// ---- GlobalTextList.TcGTLO
TEXTLIST GlobalTextList
  6525 = ' '
  3937 = '      Suction'
  4564 = '     KR5 Magnet'
  5885 = '     Magnet'
  1846 = ' Suction'
  271 = '%s'
  243 = '+'
  1867 = '-'
  4558 = '1-100'
  645 = '10'
  4817 = '100-200'
  551 = '1000'
  201 = '1001'
  301 = '1002'
  663 = '1003'
  224 = '1004'
  174 = '1005'
  178 = '1006'
  933 = '1007'
  532 = '1008'
  34 = '1027'
  349 = '1028'
  986 = '1029'
  837 = '1030'
  751 = '1031'
  65 = '1032'
  93 = '1033'
  410 = '1034'
  763 = '1035'
  289 = '1036'
  454 = '1037'
  54 = '1038'
  692 = '1039'
  219 = '1040'
  822 = '1041'
  60 = '1042'
  614 = '1222'
  158 = '130'
  797 = '2.00'
  613 = '20'
  808 = '200'
  239 = '201'
  348 = '202'
  665 = '203'
  496 = '204'
  79 = '205'
  623 = '206'
  342 = '207'
  798 = '208'
  844 = '209'
  393 = '210'
  250 = '211'
  526 = '212'
  221 = '213'
  611 = '214'
  925 = '215'
  371 = '216'
  469 = '217'
  431 = '218'
  816 = '219'
  447 = '220'
  514 = '221'
  909 = '222'
  626 = '2221'
  7 = '223'
  817 = '224'
  341 = '225'
  3095 = '226'
  3222 = '227'
  1709 = '228'
  2374 = '229'
  985 = '230'
  2478 = '231'
  5328 = '245'
  5414 = '246'
  5250 = '247'
  836 = '300'
  444 = '301'
  863 = '302'
  136 = '303'
  503 = '304'
  148 = '305'
  196 = '30518'
  888 = '306'
  951 = '307'
  2719 = '7'
  987 = '993'
  157 = '994'
  133 = '995'
  412 = '996'
  103 = '997'
  549 = '998'
  772 = '999'
  730 = 'A1'
  855 = 'A1 Filled'
  1134 = 'A1 Sensor'
  1013 = 'A1 to JIG A'
  3517 = 'A1/B1'
  761 = 'A1_FG'
  1763 = 'A2'
  809 = 'A2 Sensor'
  1844 = 'A2 to JIG A'
  295 = 'A2/B2'
  200 = 'A3'
  891 = 'A3 Sensor'
  1636 = 'A3 to JIG A'
  279 = 'A3/B3'
  1957 = 'A4'
  939 = 'A4 Sensor'
  516 = 'A4 to JIG A'
  1942 = 'A4/B4'
  3137 = 'A45'
  46 = 'A5'
  1043 = 'A5 Sensor'
  357 = 'A5 to JIG A'
  2399 = 'A5/B5'
  426 = 'Admin'
  49 = 'ADMIN'
  1229 = 'Air Pressure'
  741 = 'Alarm Stop'
  1217 = 'Appl Run'
  1955 = 'Aut'
  832 = 'Auto Mode Run Production'
  1054 = 'B1'
  540 = 'B1 or'
  567 = 'B1 Sensor'
  3022 = 'B1 to JIG A'
  1677 = 'B2'
  778 = 'B2 Sensor'
  3456 = 'B2 to JIG A'
  1682 = 'B3'
  1188 = 'B3 Sensor'
  2731 = 'B3 to JIG A'
  1139 = 'B4'
  245 = 'B4 Sensor'
  1366 = 'B4 to JIG A'
  1154 = 'B5'
  921 = 'B5 Sensor'
  682 = 'B5 to JIG A'
  1172 = 'Back'
  1818 = 'Basket A'
  191 = 'Basket B'
  795 = 'Bot 1'
  1887 = 'Bot 2'
  1276 = 'Bot 3'
  1810 = 'Bot 4'
  979 = 'Bot 5'
  1585 = 'Bot 6'
  1939 = 'Bot 7'
  4142 = 'Buzzer Mute'
  3618 = 'Bypass KR1 will cause danger to the workcell. \nYES to confirm\nproceed with own risk !'
  6774 = 'Bypass KR2 will cause danger to the workcell, Please confirm'
  82 = 'Bypass KR2 will cause danger to the workcell. \nYES to confirm\nproceed with own risk !'
  1492 = 'Bypass KR2 will cause danger to the workcell. \nYES to confirm, proceed with own risk !'
  1503 = 'Bypass KR2 will cause danger to the workcell. Proceed with own risk'
  28 = 'Bypass KR2 will cause danger to the workcell. Proceed with own risk !'
  385 = 'Bypass KR2 will cause danger to the workcell. YES to confirm, proceed with own risk !'
  4768 = 'Bypass KR2 will cause danger to the workcell.YES to proceed with own risk !'
  504 = 'Bypass KR4 will cause danger to the workcell. \nYES to confirm\nproceed with own risk !'
  483 = 'C.Rack 21'
  270 = 'C.Rack B1'
  1020 = 'C.Rack B2'
  311 = 'C.Rack B3'
  517 = 'C.Rack B4'
  1209 = 'C.Rack B5'
  1063 = 'C.Rack B6'
  1249 = 'C.Rack B7'
  515 = 'C.Rack M1'
  690 = 'C.Rack M2'
  427 = 'C.Rack M3'
  1226 = 'C.Rack M4'
  1052 = 'C.Rack M5'
  530 = 'C.Rack M6'
  1495 = 'C.Rack M7'
  364 = 'C.Rack T1'
  1341 = 'C.Rack T2'
  321 = 'C.Rack T3'
  1219 = 'C.Rack T4'
  397 = 'C.Rack T5'
  1314 = 'C.Rack T6'
  637 = 'C.Rack T7'
  1328 = 'C010'
  2038 = 'Cancel'
  2814 = 'Clean Torch'
  3342 = 'Clear Error'
  3039 = 'Complete'
  1015 = 'Conf Mess'
  2439 = 'Confirm Reset Production Sequance ?'
  3216 = 'Confirm RESET Production Sequance ?'
  602 = 'Connect IFRACK'
  1182 = 'Connect IFRack'
  918 = 'Conveyor Full'
  263 = 'Cool Rack T1'
  97 = 'Cooling Rack'
  1330 = 'Cooling Time'
  1050 = 'COSMO'
  389 = 'COSMO FAIL'
  3699 = 'Cosmo Fail'
  1107 = 'COSMO Fail Unit : '
  381 = 'COSMO NO OK'
  338 = 'COSMO OK'
  40 = 'COSMO PASS'
  2525 = 'COSMO Pass'
  197 = 'Cosmo Pass'
  2755 = 'COSMO Pass Unit :'
  45 = 'COSMO Ready'
  1270 = 'COSMO Run'
  1562 = 'COSMO Standby'
  2340 = 'CR'
  956 = 'CR01'
  3889 = 'CR01  COSMO'
  3781 = 'CR01 COSMO'
  2044 = 'CR01 JIG'
  2799 = 'CR010'
  1537 = 'CR011'
  536 = 'CR02'
  2652 = 'CR02 COSMO'
  2480 = 'CR02 JIG'
  98 = 'CR02 to COSMO'
  1900 = 'CR03'
  2621 = 'CR03 COSMO'
  6608 = 'CR03 COSMO227'
  1956 = 'CR03 JIG'
  2471 = 'CR04'
  1816 = 'CR04 COSMO'
  4062 = 'CR04 JIG'
  597 = 'CR05'
  718 = 'CR05 COSMO'
  2378 = 'CR05 JIG'
  932 = 'CR06'
  1198 = 'CR06 COSMO'
  897 = 'CR06 JIG'
  1838 = 'CR07'
  1322 = 'CR07 COSMO'
  1577 = 'CR07 JIG'
  1698 = 'CR070 COSMO'
  315 = 'CR08'
  3906 = 'CR08 COSMO'
  1342 = 'CR08 JIG'
  1470 = 'CR09'
  1716 = 'CR09 COSMO'
  3068 = 'CR09 JIG'
  1578 = 'CR1 to COSMO'
  675 = 'CR10'
  459 = 'CR10 COSMO'
  651 = 'CR10 JIG'
  2872 = 'CR10 to COSMO'
  2858 = 'CR11'
  2361 = 'CR11 COSMO'
  1703 = 'CR11 JIG'
  706 = 'CR11 to COSMO'
  2165 = 'CR12'
  1881 = 'CR12 COSMO'
  3782 = 'CR12 JIG'
  997 = 'CR12 to COSMO'
  2650 = 'CR13'
  1277 = 'CR13 COSMO'
  6430 = 'CR13 JIG'
  2293 = 'CR13 to COSMO'
  2373 = 'CR14 COSMO'
  1649 = 'CR14 to COSMO'
  1874 = 'CR15'
  5638 = 'CR15 COSMO'
  5944 = 'CR15 JIG'
  2382 = 'CR16'
  527 = 'CR16 COSMO'
  3201 = 'CR16 JIG'
  1111 = 'CR17'
  5326 = 'CR17 COSMO'
  120 = 'CR17 JIG'
  1765 = 'CR18'
  1780 = 'CR18 COSMO'
  2849 = 'CR18 JIG'
  1690 = 'CR19'
  2783 = 'CR19 COSMO'
  3793 = 'CR19 JIG'
  1498 = 'CR2 to COSMO'
  1862 = 'CR2. JIG'
  229 = 'CR20'
  4286 = 'CR20 COSMO'
  3843 = 'CR20 JIG'
  2764 = 'CR21'
  3780 = 'CR21 COSMO'
  4896 = 'CR21 JIG'
  1336 = 'CR3 to COSMO'
  1901 = 'CR4 to COSMO'
  1505 = 'CR5 to COSMO'
  3031 = 'CR6 to COSMO'
  276 = 'CR7 to COSMO'
  2514 = 'CR8 to COSMO'
  2642 = 'CR9 to COSMO'
  1204 = 'Cycle Count'
  1027 = 'Cycle Count :'
  172 = 'Daily Count'
  848 = 'Daily Count :'
  2224 = 'Daily Output :'
  4545 = 'Door Close'
  2536 = 'Drive Off'
  664 = 'Drive On'
  35 = 'Emergency Stop All'
  2372 = 'End Conveyor'
  1981 = 'End FG1'
  983 = 'Engineer'
  1852 = 'Error'
  1405 = 'Ext'
  1574 = 'Ext Start'
  96 = 'Face A'
  857 = 'Face B'
  774 = 'Fail Unit : '
  4436 = 'FaiUnit : '
  624 = 'FG'
  32 = 'FG Last Pack Pos'
  2718 = 'FG1 1'
  4083 = 'FG1 Po157'
  2184 = 'FG1 Po1s84'
  2502 = 'FG1 Po1s85'
  5123 = 'FG1 Po1s86'
  2804 = 'FG1 Po1s93'
  1855 = 'FG1 Pos1'
  1406 = 'FG1 Pos10'
  4148 = 'FG1 Pos100'
  566 = 'FG1 Pos101'
  2929 = 'FG1 Pos102'
  4304 = 'FG1 Pos103'
  1699 = 'FG1 Pos104'
  4284 = 'FG1 Pos105'
  1663 = 'FG1 Pos106'
  3032 = 'FG1 Pos107'
  5412 = 'FG1 Pos108'
  2069 = 'FG1 Pos109'
  4509 = 'FG1 Pos11'
  3003 = 'FG1 Pos110'
  5981 = 'FG1 Pos111'
  3826 = 'FG1 Pos112'
  6305 = 'FG1 Pos113'
  4145 = 'FG1 Pos114'
  2798 = 'FG1 Pos115'
  5872 = 'FG1 Pos116'
  1125 = 'FG1 Pos117'
  3736 = 'FG1 Pos118'
  5178 = 'FG1 Pos119'
  2721 = 'FG1 Pos12'
  4463 = 'FG1 Pos120'
  634 = 'FG1 Pos121'
  5542 = 'FG1 Pos122'
  5185 = 'FG1 Pos123'
  1664 = 'FG1 Pos124'
  2535 = 'FG1 Pos125'
  2532 = 'FG1 Pos126'
  4938 = 'FG1 Pos127'
  6511 = 'FG1 Pos128'
  1615 = 'FG1 Pos129'
  995 = 'FG1 Pos13'
  4585 = 'FG1 Pos130'
  3268 = 'FG1 Pos131'
  1968 = 'FG1 Pos132'
  6219 = 'FG1 Pos133'
  5372 = 'FG1 Pos134'
  1262 = 'FG1 Pos135'
  5169 = 'FG1 Pos136'
  6201 = 'FG1 Pos137'
  5235 = 'FG1 Pos138'
  3852 = 'FG1 Pos139'
  3497 = 'FG1 Pos14'
  5668 = 'FG1 Pos140'
  6182 = 'FG1 Pos141'
  4599 = 'FG1 Pos142'
  3554 = 'FG1 Pos143'
  839 = 'FG1 Pos144'
  208 = 'FG1 Pos145'
  1520 = 'FG1 Pos146'
  1580 = 'FG1 Pos147'
  3817 = 'FG1 Pos148'
  3964 = 'FG1 Pos149'
  2490 = 'FG1 Pos15'
  850 = 'FG1 Pos150'
  3387 = 'FG1 Pos151'
  317 = 'FG1 Pos152'
  3953 = 'FG1 Pos153'
  1552 = 'FG1 Pos154'
  4104 = 'FG1 Pos155'
  2467 = 'FG1 Pos156'
  4670 = 'FG1 Pos158'
  2341 = 'FG1 Pos159'
  1512 = 'FG1 Pos16'
  1485 = 'FG1 Pos160'
  5555 = 'FG1 Pos161'
  5825 = 'FG1 Pos162'
  4681 = 'FG1 Pos163'
  4823 = 'FG1 Pos164'
  5092 = 'FG1 Pos165'
  1041 = 'FG1 Pos166'
  4077 = 'FG1 Pos167'
  2126 = 'FG1 Pos168'
  4672 = 'FG1 Pos169'
  3046 = 'FG1 Pos17'
  1312 = 'FG1 Pos170'
  1300 = 'FG1 Pos171'
  2684 = 'FG1 Pos172'
  5600 = 'FG1 Pos173'
  4222 = 'FG1 Pos174'
  3422 = 'FG1 Pos175'
  5984 = 'FG1 Pos176'
  5270 = 'FG1 Pos177'
  5089 = 'FG1 Pos178'
  1354 = 'FG1 Pos179'
  303 = 'FG1 Pos18'
  3565 = 'FG1 Pos180'
  1144 = 'FG1 Pos181'
  2064 = 'FG1 Pos182'
  4513 = 'FG1 Pos183'
  810 = 'FG1 Pos184'
  5562 = 'FG1 Pos185'
  2178 = 'FG1 Pos186'
  4633 = 'FG1 Pos187'
  1595 = 'FG1 Pos188'
  1236 = 'FG1 Pos189'
  2725 = 'FG1 Pos19'
  2883 = 'FG1 Pos190'
  70 = 'FG1 Pos191'
  2370 = 'FG1 Pos192'
  3987 = 'FG1 Pos193'
  953 = 'FG1 Pos194'
  4997 = 'FG1 Pos195'
  1045 = 'FG1 Pos196'
  4749 = 'FG1 Pos197'
  2703 = 'FG1 Pos198'
  4116 = 'FG1 Pos199'
  233 = 'FG1 Pos2'
  2491 = 'FG1 Pos20'
  2255 = 'FG1 Pos200'
  1776 = 'FG1 Pos21'
  1227 = 'FG1 Pos22'
  2963 = 'FG1 Pos23'
  1654 = 'FG1 Pos24'
  3123 = 'FG1 Pos25'
  557 = 'FG1 Pos26'
  3705 = 'FG1 Pos27'
  688 = 'FG1 Pos28'
  3637 = 'FG1 Pos29'
  1573 = 'FG1 Pos3'
  1164 = 'FG1 Pos30'
  1788 = 'FG1 Pos31'
  4210 = 'FG1 Pos32'
  3810 = 'FG1 Pos33'
  3318 = 'FG1 Pos34'
  2449 = 'FG1 Pos35'
  3264 = 'FG1 Pos36'
  3507 = 'FG1 Pos37'
  2001 = 'FG1 Pos38'
  3057 = 'FG1 Pos39'
  599 = 'FG1 Pos4'
  2071 = 'FG1 Pos40'
  2161 = 'FG1 Pos41'
  2496 = 'FG1 Pos42'
  955 = 'FG1 Pos43'
  3060 = 'FG1 Pos44'
  1806 = 'FG1 Pos45'
  4323 = 'FG1 Pos46'
  3819 = 'FG1 Pos47'
  2191 = 'FG1 Pos48'
  1555 = 'FG1 Pos49'
  1337 = 'FG1 Pos5'
  3357 = 'FG1 Pos50'
  555 = 'FG1 Pos51'
  1652 = 'FG1 Pos52'
  3905 = 'FG1 Pos53'
  1181 = 'FG1 Pos54'
  199 = 'FG1 Pos55'
  2461 = 'FG1 Pos56'
  76 = 'FG1 Pos57'
  622 = 'FG1 Pos58'
  3257 = 'FG1 Pos59'
  3131 = 'FG1 Pos6'
  2727 = 'FG1 Pos60'
  615 = 'FG1 Pos61'
  5038 = 'FG1 Pos62'
  1246 = 'FG1 Pos63'
  4226 = 'FG1 Pos64'
  4198 = 'FG1 Pos65'
  1908 = 'FG1 Pos66'
  981 = 'FG1 Pos67'
  1234 = 'FG1 Pos68'
  3745 = 'FG1 Pos69'
  2629 = 'FG1 Pos7'
  1407 = 'FG1 Pos70'
  4162 = 'FG1 Pos71'
  3749 = 'FG1 Pos72'
  4799 = 'FG1 Pos73'
  2591 = 'FG1 Pos74'
  2075 = 'FG1 Pos75'
  2352 = 'FG1 Pos76'
  5078 = 'FG1 Pos77'
  2641 = 'FG1 Pos78'
  4011 = 'FG1 Pos79'
  1628 = 'FG1 Pos8'
  3927 = 'FG1 Pos80'
  600 = 'FG1 Pos81'
  4659 = 'FG1 Pos82'
  2512 = 'FG1 Pos83'
  5039 = 'FG1 Pos84'
  4204 = 'FG1 Pos85'
  4255 = 'FG1 Pos86'
  2310 = 'FG1 Pos87'
  1762 = 'FG1 Pos88'
  1231 = 'FG1 Pos89'
  799 = 'FG1 Pos9'
  625 = 'FG1 Pos90'
  1131 = 'FG1 Pos91'
  3965 = 'FG1 Pos92'
  2797 = 'FG1 Pos93'
  4004 = 'FG1 Pos94'
  2531 = 'FG1 Pos95'
  1317 = 'FG1 Pos96'
  577 = 'FG1 Pos97'
  4568 = 'FG1 Pos98'
  3794 = 'FG1 Pos99'
  3834 = 'Gas Pressure'
  3918 = 'Get Layer Pad'
  1841 = 'Get Magnet'
  4355 = 'Get Suction'
  1420 = 'Go Home'
  3858 = 'Halt   Production'
  2679 = 'Halt Production'
  362 = 'IFRack Online'
  752 = 'IFRackOnline'
  978 = 'IFRack_A1'
  838 = 'IFRack_A15'
  678 = 'IFRack_A2'
  384 = 'IFRack_A3'
  198 = 'IFRack_A4'
  942 = 'IFRack_A5'
  998 = 'IFRack_B1'
  587 = 'IFRack_B2'
  954 = 'IFRack_B3'
  660 = 'IFRack_B4'
  84 = 'IFRack_B5'
  12 = 'IFRack_Online'
  2266 = 'In Home'
  731 = 'Infeed Rack'
  2084 = 'IO Act'
  1875 = 'IO Act Confg'
  552 = 'IO ActConf'
  333 = 'IPC Input'
  392 = 'IPC Output'
  299 = 'Is Magnet attached on KR1 ?'
  1156 = 'Is Suction Cup attached on KR1 ?'
  926 = 'JIG'
  2011 = 'JIG '
  636 = 'JIG A'
  240 = 'JIG A Clamp'
  1040 = 'JIG A Complete'
  512 = 'JIG A Ready'
  963 = 'JIG A Release'
  1360 = 'JIG A Standby'
  633 = 'JIG A to JIG B'
  961 = 'JIG A to Welding'
  524 = 'JIG A Welding'
  506 = 'JIG AControl'
  1687 = 'JIG B'
  14 = 'JIG B Clamp'
  500 = 'JIG B Ready'
  872 = 'JIG B Release'
  101 = 'JIG B Standby'
  2243 = 'JIG B to TT'
  1564 = 'JIG B to Welding'
  1203 = 'JIG B Welding'
  253 = 'JIG C'
  281 = 'JIG C Clamp'
  1053 = 'JIG C Ready'
  31 = 'JIG C Release'
  672 = 'JIG C Standby'
  2350 = 'Jig C to CR1'
  821 = 'Jig C to CR2'
  448 = 'Jig C to CR3'
  2012 = 'Jig C to CR4'
  2466 = 'Jig C to CR5'
  1481 = 'JIG C to Welding'
  800 = 'JIG C Welding'
  631 = 'JIG Control'
  2104 = 'Job Fail'
  1625 = 'Job Fail Sig'
  38 = 'Job Fail Signal'
  130 = 'K51 Magnet'
  267 = 'KR1'
  5061 = 'KR1 Bypass'
  966 = 'KR1 E.Stop'
  104 = 'KR1 EOAT '
  3474 = 'KR1 Magnet'
  6686 = 'KR1 Suction'
  424 = 'KR2'
  4276 = 'KR2 Bypass'
  677 = 'KR2 E.Stop'
  300 = 'KR3'
  3795 = 'KR3 Bypass'
  87 = 'KR3 E.Stop'
  886 = 'KR4'
  6395 = 'KR4 Bypass'
  180 = 'KR4 E.Stop'
  344 = 'KR5'
  533 = 'KR5 E.Stop'
  6338 = 'KR5 Magnet'
  5526 = 'KR5 Suction'
  347 = 'Kuka Robot 1'
  425 = 'Kuka Robot 2'
  584 = 'Kuka Robot 3'
  578 = 'Kuka Robot 4'
  545 = 'Kuka Robot 5'
  588 = 'L+ogin'
  6417 = 'Layer pad '
  6940 = 'Layer pad 0 is filled'
  5899 = 'Layer pad 1'
  1393 = 'Layer pad 10'
  4215 = 'Layer pad 2'
  6818 = 'Layer pad 3'
  6716 = 'Layer pad 4'
  3289 = 'Layer pad 5'
  884 = 'Layer pad 6'
  1910 = 'Layer pad 7'
  4729 = 'Layer pad 8'
  4447 = 'Layer pad 9'
  2585 = 'Login'
  1296 = 'Logout'
  118 = 'Magnet'
  1396 = 'Main'
  2380 = 'Manual Mode'
  831 = 'Manual Sequence'
  390 = 'Mid 1'
  1187 = 'Mid 2'
  468 = 'Mid 3'
  312 = 'Mid 4'
  812 = 'Mid 5'
  736 = 'Mid 6'
  585 = 'Mid 7'
  435 = 'Minutes'
  2103 = 'Move Enable'
  703 = 'Next Sequence'
  1496 = 'Next Step'
  737 = 'NO'
  3008 = 'None'
  3419 = 'OK'
  57 = 'On Path'
  4034 = 'Online'
  3383 = 'Operator'
  2438 = 'Pass unit :'
  667 = 'Password :'
  548 = 'Peri Rdy'
  2043 = 'PGNO Fbit'
  1590 = 'PGNO Parity'
  2948 = 'PGNO Req'
  1922 = 'PGNO Valid'
  892 = 'Pick Muffler'
  732 = 'Pick Rework'
  1362 = 'Pos IF A1'
  502 = 'Pos IF A2'
  1324 = 'Pos IF A3'
  2368 = 'Pos IF A4'
  3079 = 'Pos IF A5'
  1685 = 'Pos IF B1'
  3694 = 'Pos IF B2'
  316 = 'Pos IF B3'
  1906 = 'Pos IF B4'
  1812 = 'Pos IF B5'
  434 = 'Pro Act'
  2309 = 'Pro Move'
  2516 = 'Programme Selection'
  2010 = 'RC Rdy1'
  451 = 'Ready'
  215 = 'Reject In'
  261 = 'Reject Out'
  1717 = 'Remove Magnet'
  1617 = 'Remove Suction'
  419 = 'Reset'
  2295 = 'Reset All KR'
  1683 = 'Reset All Kuka'
  2232 = 'Reset Production'
  2692 = 'ResetStop All'
  2339 = 'Restart Step'
  2188 = 'Rework Done'
  1082 = 'Rework Empty'
  1213 = 'Rework In'
  2222 = 'Rework In A'
  2244 = 'Rework In B'
  1647 = 'Rework Standby'
  616 = 'Rework Unit'
  2962 = 'Rework Unit : '
  562 = 'RM79 / KR1'
  4244 = 'Robot '
  2294 = 'Robot Configuration'
  139 = 'Run '
  1998 = 'Run   Production'
  2004 = 'Run Production'
  1349 = 'RUN Sequence'
  1517 = 'Run Sequence'
  768 = 'Run Steep'
  1964 = 'Run Step'
  3044 = 'RW'
  165 = 'RW75 / KR2'
  147 = 'RW75 / KR3'
  2065 = 'RW76 / KR1'
  2092 = 'RW76 / KR5'
  225 = 'RW77 / KR2'
  914 = 'RW77 / KR3'
  1928 = 'RW78 / KR4'
  1290 = 'RW79 / KR1'
  851 = 'RW79 / KR5'
  370 = 'Seconds'
  1089 = 'Set Time'
  1540 = 'Standby'
  652 = 'Start Time'
  2057 = 'Stop'
  959 = 'Stop Mess'
  717 = 'Stop Production'
  1395 = 'Suction'
  574 = 'T.Torch Clamp'
  988 = 'T.Torch Complaete'
  161 = 'T.Torch Complete'
  58 = 'T.Torch Run'
  814 = 'T.Torch Standby'
  2379 = 'T1'
  2856 = 'T2'
  100 = 'Toggle IFRack'
  903 = 'Top  3'
  819 = 'Top 1'
  890 = 'Top 2'
  1673 = 'Top 3'
  1161 = 'Top 4'
  1389 = 'Top 5'
  1678 = 'Top 6'
  666 = 'Top 7'
  525 = 'Torch Clean'
  3519 = 'Torch Cleaning'
  700 = 'TT to JIG C'
  3513 = 'Turn Ready'
  288 = 'Turn to A'
  906 = 'Turn to B'
  2099 = 'Twin Torch'
  2336 = 'Use Saf'
  842 = 'User :'
  1869 = 'User Saf'
  4844 = 'v\nLayer pad 5'
  411 = 'V.B Sensor'
  5411 = 'v7'
  991 = 'VB to Jig C'
  879 = 'VB to JIG C'
  1916 = 'Weekly Count :'
  1946 = 'Weekly Output :'
  2921 = 'Welcome, '
  523 = 'Welcome, Admin'
  3045 = 'Welcome, Engineer'
  1710 = 'Welcome, Jackson'
  3796 = 'Welcome, Operator'
  3014 = 'Welding Mode'
  1190 = 'Work Cell 1'
  2233 = 'Work Cell 1 (Under Maintainance)'
  1741 = 'Work Cell 1 (Under Reconfiguration)'
  3807 = 'YES'
  2314 = '_'
END_TEXTLIST

// ---- POUs/User.TcTLO
TEXTLIST User
  0 = 'None'
  1 = 'Engineer'
  2 = 'Technician'
  3 = 'Operator'
   = ''
END_TEXTLIST

// ---- VISUs/Dialog/MSG_BOX_RESET.TcVIS
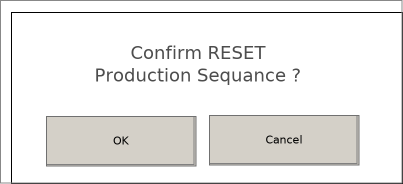
VISUALIZATION MSG_BOX_RESET  // 403x184
    RoundedRectangle (11,12 392x172)
    Button (46,116 150x50), "OK"
        OnMouseClick: execute {
            LOGFILE( sLogEvent	 := MSG.EVENT_BTN,
            		 sLogComp	 := MSG.COMP_HMI,
            		 sLogAction	 := MSG.ACTION_RESET,
            		 logFlag	 := TRUE);
            AUTO_MODE.Reset_seq_btn:= true;
        }
        OnMouseClick: CloseDialog Dialog=MSG_BOX_RESET, Result=OK, NumpadKeypadSet=True
    Button (209,115 150x50), "Cancel"
        OnMouseClick: CloseDialog Dialog=MSG_BOX_RESET, Result=Cancel, NumpadKeypadSet=True
    Label (80,20 236x88), "Confirm RESET Production Sequance ?"
END_VISUALIZATION

// ---- VISUs/Dialog/MSG_EOAT.TcVIS
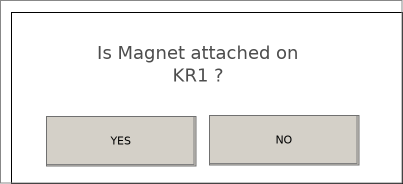
VISUALIZATION MSG_EOAT  // 403x184
    RoundedRectangle (11,12 392x172)
    Button (46,116 150x50), "YES"
        OnMouseClick: execute { GVL.KR1_EOAT_FILL:= TRUE; GVL.KR1_EOAT_SUCTION:= FALSE; }
        OnMouseClick: CloseDialog Dialog=MSG_EOAT, Result=Yes, NumpadKeypadSet=True
    Button (209,115 150x50), "NO"
        OnMouseClick: execute { GVL.KR1_EOAT_FILL:= FALSE; }
        OnMouseClick: CloseDialog Dialog=MSG_EOAT, Result=No, NumpadKeypadSet=True
    Label (80,20 236x88), "Is Magnet attached on KR1 ?"
END_VISUALIZATION

// ---- VISUs/Dialog/MSG_EOAT_SUCTION.TcVIS
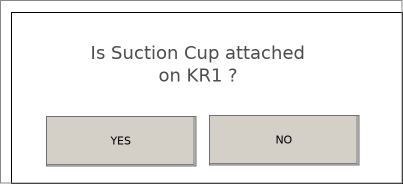
VISUALIZATION MSG_EOAT_SUCTION  // 403x184
    RoundedRectangle (11,12 392x172)
    Button (46,116 150x50), "YES"
        OnMouseClick: execute { GVL.KR1_EOAT_FILL:= FALSE; GVL.KR1_EOAT_SUCTION:= TRUE; }
        OnMouseClick: CloseDialog Dialog=MSG_EOAT_SUCTION, Result=Yes, NumpadKeypadSet=True
    Button (209,115 150x50), "NO"
        OnMouseClick: execute { GVL.KR1_EOAT_SUCTION:= FALSE; }
        OnMouseClick: CloseDialog Dialog=MSG_EOAT_SUCTION, Result=No, NumpadKeypadSet=True
    Label (80,20 236x88), "Is Suction Cup attached on KR1 ?"
END_VISUALIZATION

// ---- VISUs/Dialog/MSG_KR2_BP.TcVIS
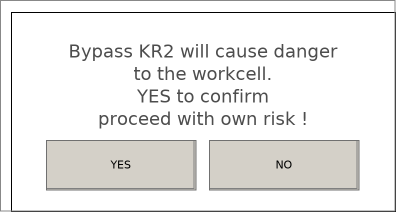
VISUALIZATION MSG_KR2_BP  // 396x212
    RoundedRectangle (11,12 385x200)
    Button (46,140 150x50), "YES"
        OnMouseClick: CloseDialog Dialog=MSG_KR2_BP, Result=Yes, NumpadKeypadSet=True
        OnMouseClick: execute { GVL.KR2_bypass := TRUE; }
    Button (209,140 150x50), "NO"
        OnMouseClick: execute { GVL.KR2_bypass := FALSE; }
        OnMouseClick: CloseDialog Dialog=MSG_KR2_BP, Result=No, NumpadKeypadSet=True
    Label (55,30 296x110), "Bypass KR2 will cause danger to the workcell. YES to confirm proceed with own risk !"
END_VISUALIZATION

// ---- VISUs/Dialog/MSG_KR4_BP.TcVIS
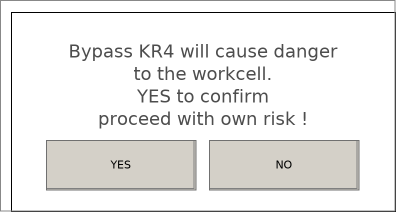
VISUALIZATION MSG_KR4_BP  // 396x212
    RoundedRectangle (11,12 385x200)
    Button (46,140 150x50), "YES"
        OnMouseClick: CloseDialog Dialog=MSG_KR4_BP, Result=Yes, NumpadKeypadSet=True
        OnMouseClick: execute { GVL.KR4_bypass := TRUE; }
    Button (209,140 150x50), "NO"
        OnMouseClick: execute { GVL.KR4_bypass := FALSE; }
        OnMouseClick: CloseDialog Dialog=MSG_KR4_BP, Result=No, NumpadKeypadSet=True
    Label (55,30 296x110), "Bypass KR4 will cause danger to the workcell. YES to confirm proceed with own risk !"
END_VISUALIZATION

// ---- VISUs/Dialog/MSG_KR1_BP.TcVIS
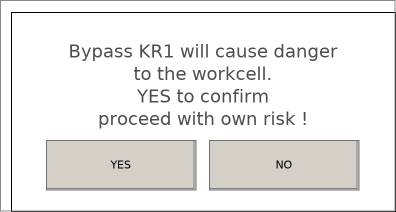
VISUALIZATION MSG_KR1_BP  // 396x212
    RoundedRectangle (11,12 385x200)
    Button (46,140 150x50), "YES"
        OnMouseClick: CloseDialog Dialog=MSG_KR1_BP, Result=Yes, NumpadKeypadSet=True
        OnMouseClick: execute { GVL.KR1_bypass := TRUE; }
    Button (209,140 150x50), "NO"
        OnMouseClick: execute { GVL.KR1_bypass := FALSE; }
        OnMouseClick: CloseDialog Dialog=MSG_KR1_BP, Result=No, NumpadKeypadSet=True
    Label (55,30 296x110), "Bypass KR1 will cause danger to the workcell. YES to confirm proceed with own risk !"
END_VISUALIZATION

// ---- VISUs/Dialog/MSG_KR3_BP.TcVIS
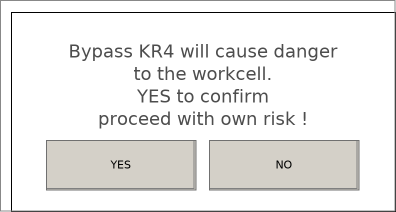
VISUALIZATION MSG_KR3_BP  // 396x212
    RoundedRectangle (11,12 385x200)
    Button (46,140 150x50), "YES"
        OnMouseClick: CloseDialog Dialog=MSG_KR3_BP, Result=Yes, NumpadKeypadSet=True
        OnMouseClick: execute { GVL.KR3_bypass := TRUE; }
    Button (209,140 150x50), "NO"
        OnMouseClick: execute { GVL.KR3_bypass := FALSE; }
        OnMouseClick: CloseDialog Dialog=MSG_KR3_BP, Result=No, NumpadKeypadSet=True
    Label (55,30 296x110), "Bypass KR4 will cause danger to the workcell. YES to confirm proceed with own risk !"
END_VISUALIZATION

// ---- VISUs/Footer_Main.TcVIS
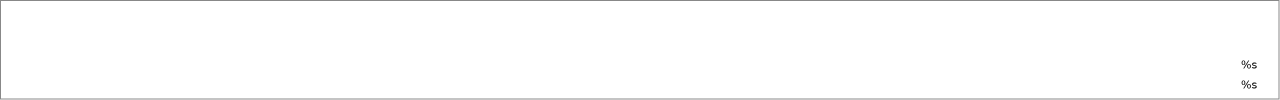
VISUALIZATION Footer_Main  // 1280x100
    Textfield (1160,70 100x30), "%s", text variable: MAIN.fb_TimeStamp.SystemDate
    Textfield (1160,50 100x30), "%s", text variable: MAIN.fb_TimeStamp.SystemTime
END_VISUALIZATION

// ---- VISUs/Footer_Back.TcVIS
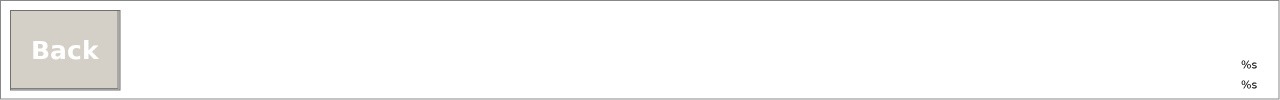
VISUALIZATION Footer_Back  // 1280x100
    Textfield (1160,70 100x30), "%s", text variable: MAIN.fb_TimeStamp.SystemDate
    Textfield (1160,50 100x30), "%s", text variable: MAIN.fb_TimeStamp.SystemTime
    Button (10,10 110x80), "Back"
        OnMouseClick: execute {
            LOGFILE( sLogEvent	 := MSG.EVENT_BTN,
            		 sLogComp	 := MSG.COMP_HMI,
            		 sLogAction	 := MSG.ACTION_BACK,
            	 	 logFlag	 := TRUE);
        }
        OnMouseClick: change screen: PAGE_MAIN
END_VISUALIZATION

// ---- VISUs/Header.TcVIS
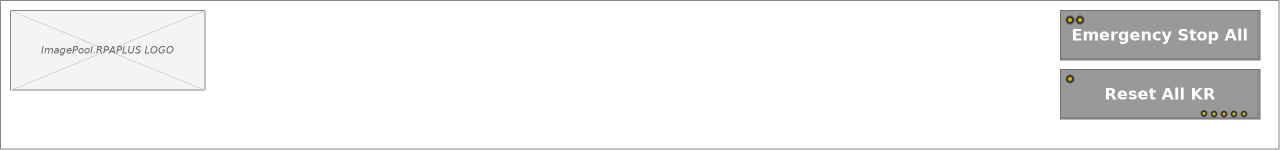
VISUALIZATION Header  // 1280x150
    Button (1060,10 200x50), "Emergency Stop All", pressed state: MAIN.btnSoftEstop
        toggle MAIN.btnSoftEstop
        OnMouseClick: execute {
            LOGFILE( sLogEvent	 := MSG.EVENT_BTN,
            		 sLogComp	 := MSG.COMP_HMI,
            		 sLogAction	 := MSG.ACTION_ESTOP,
            	 	 logFlag	 := TRUE);
        }
    Image (10,10 195x80), image: ImagePool.RPAPLUS LOGO
    Button (1060,69 200x50), "Reset All KR", pressed state: MAIN.btn_Reset or MAIN.Reset_State
        tap MAIN.btn_Reset
        OnMouseClick: execute {
            LOGFILE( sLogEvent	 := MSG.EVENT_BTN,
            		 sLogComp	 := MSG.COMP_HMI,
            		 sLogAction	 := MSG.ACTION_RESET_KUKA,
            	 	 logFlag	 := TRUE);
        }
    Lamp1 (1065,74 10x10), variable: MAIN.Reset_State, style: Lamp-Lamp1-Yellow
    Lamp1 (1200,109 8x9), variable: KR5.KR_ProgReady, style: Lamp-Lamp1-Yellow
    Lamp1 (1240,109 8x10), variable: KR1.KR_ProgReady, style: Lamp-Lamp1-Yellow
    Lamp1 (1230,109 8x10), variable: KR4.KR_ProgReady, style: Lamp-Lamp1-Yellow
    Lamp1 (1220,109 8x10), variable: KR2.KR_ProgReady, style: Lamp-Lamp1-Yellow
    Lamp1 (1210,109 8x10), variable: KR3.KR_ProgReady, style: Lamp-Lamp1-Yellow
    Lamp1 (1065,15 10x10), variable: not MAIN.btnEstop, style: Lamp-Lamp1-Yellow
    Lamp1 (1075,15 10x10), variable: MAIN.btnSoftEstop, style: Lamp-Lamp1-Yellow
END_VISUALIZATION

// ---- VISUs/PAGE_InfeedRack.TcVIS
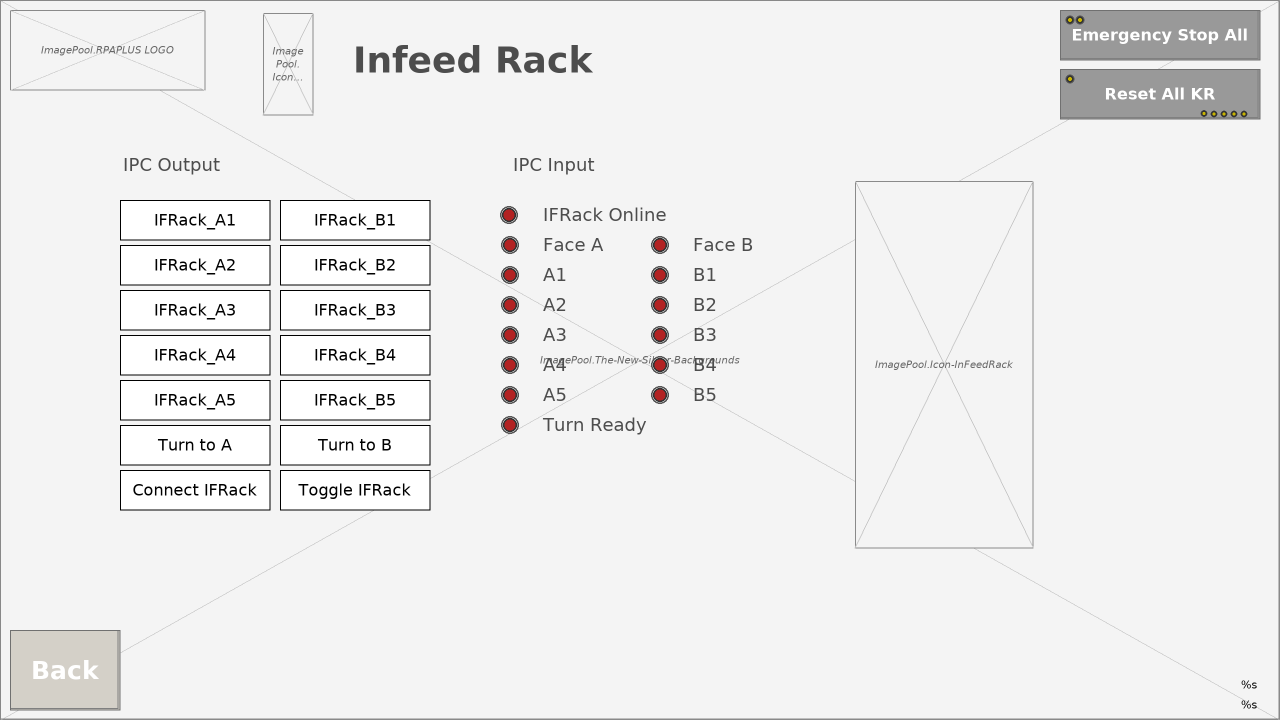
VISUALIZATION PAGE_InfeedRack  // 1280x720
    Image (0,0 1280x720), image: ImagePool.The-New-Silver-Backgrounds
    Frame (0,620 1280x100)
        shows Footer_Back()
    Frame (0,0 1280x150)
        shows Header()
    Label (350,40 300x40), "Infeed Rack"
    Label (120,150 150x30), "IPC Output"
    RoundedRectangle (120,200 150x40), "IFRack_A1"
        toggle INFEED_RACK.A1_Valve
    RoundedRectangle (120,245 150x40), "IFRack_A2"
        toggle INFEED_RACK.A2_Valve
    RoundedRectangle (120,290 150x40), "IFRack_A3"
        toggle INFEED_RACK.A3_Valve
    RoundedRectangle (120,335 150x40), "IFRack_A4"
        toggle INFEED_RACK.A4_Valve
    RoundedRectangle (120,380 150x40), "IFRack_A5"
        toggle INFEED_RACK.A5_Valve
    RoundedRectangle (280,200 150x40), "IFRack_B1"
        toggle INFEED_RACK.B1_Valve
    RoundedRectangle (280,245 150x40), "IFRack_B2"
        toggle INFEED_RACK.B2_Valve
    RoundedRectangle (280,290 150x40), "IFRack_B3"
        toggle INFEED_RACK.B3_Valve
    RoundedRectangle (280,335 150x40), "IFRack_B4"
        toggle INFEED_RACK.B4_Valve
    RoundedRectangle (280,380 150x40), "IFRack_B5"
        toggle INFEED_RACK.B5_Valve
    RoundedRectangle (120,425 150x40), "Turn to A"
        toggle INFEED_RACK.Turn_B_to_A
    RoundedRectangle (280,425 150x40), "Turn to B"
        toggle INFEED_RACK.Turn_A_to_B
    RoundedRectangle (120,470 150x40), "Connect IFRack"
        toggle INFEED_RACK.IFRack_Connect
    RoundedRectangle (280,470 150x40), "Toggle IFRack"
        tap INFEED_RACK.bstart_Write
    Label (510,150 150x30), "IPC Input"
    Label (540,380 100x30), "A5"
    Label (690,380 100x30), "B5"
    Label (540,200 130x30), "IFRack Online"
    Lamp1 (499,205 20x20), variable: INFEED_RACK.IFRack_Ready, style: Lamp-Lamp1-Red
    Lamp1 (500,235 20x20), variable: INFEED_RACK.FaceA_InWC, style: Lamp-Lamp1-Red
    Lamp1 (500,265 20x20), variable: INFEED_RACK.A1_Sensor, style: Lamp-Lamp1-Red
    Lamp1 (500,295 20x20), variable: INFEED_RACK.A2_Sensor, style: Lamp-Lamp1-Red
    Lamp1 (500,325 20x20), variable: INFEED_RACK.A3_Sensor, style: Lamp-Lamp1-Red
    Label (540,260 100x30), "A1"
    Label (540,290 100x30), "A2"
    Label (540,320 100x30), "A3"
    Label (540,350 100x30), "A4"
    Lamp1 (500,355 20x20), variable: INFEED_RACK.A4_Sensor, style: Lamp-Lamp1-Red
    Lamp1 (500,385 20x20), variable: INFEED_RACK.A5_Sensor, style: Lamp-Lamp1-Red
    Label (540,230 100x30), "Face A"
    Lamp1 (650,235 20x20), variable: INFEED_RACK.FaceB_InWC, style: Lamp-Lamp1-Red
    Lamp1 (650,265 20x20), variable: INFEED_RACK.B1_Sensor, style: Lamp-Lamp1-Red
    Lamp1 (650,295 20x20), variable: INFEED_RACK.B2_Sensor, style: Lamp-Lamp1-Red
    Lamp1 (650,325 20x20), variable: INFEED_RACK.B3_Sensor, style: Lamp-Lamp1-Red
    Label (690,260 100x30), "B1"
    Label (690,290 100x30), "B2"
    Label (690,320 100x30), "B3"
    Label (690,350 100x30), "B4"
    Lamp1 (650,355 20x20), variable: INFEED_RACK.B4_Sensor, style: Lamp-Lamp1-Red
    Lamp1 (650,385 20x20), variable: INFEED_RACK.B5_Sensor, style: Lamp-Lamp1-Red
    Label (690,230 100x30), "Face B"
    Image (263,13 50x102), image: ImagePool.Icon-InFeedRack
    Image (855,181 178x367), image: ImagePool.Icon-InFeedRack
    Lamp1 (500,415 20x20), variable: INFEED_RACK.IFRack_TurnReady, style: Lamp-Lamp1-Red
    Label (540,410 127x30), "Turn Ready"
END_VISUALIZATION

// ---- VISUs/PAGE_COSMO.TcVIS
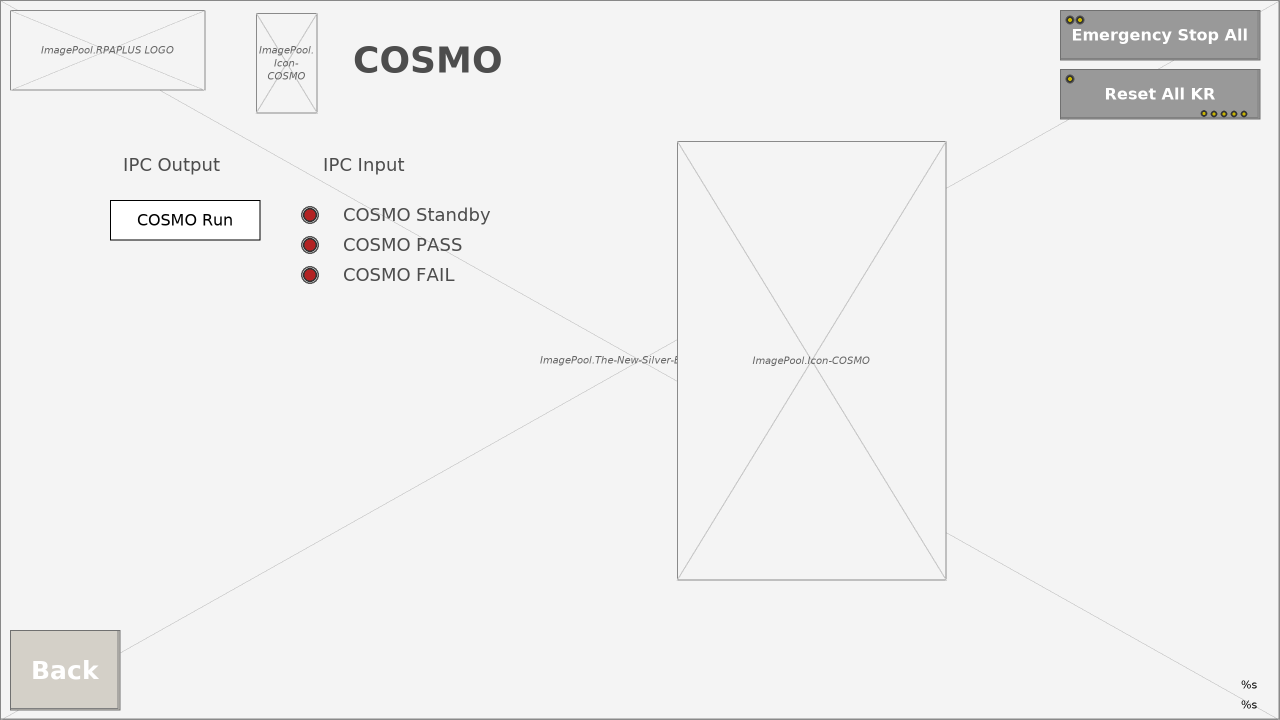
VISUALIZATION PAGE_COSMO  // 1280x720
    Image (0,0 1280x720), image: ImagePool.The-New-Silver-Backgrounds
    Frame (0,620 1280x100)
        shows Footer_Back()
    Frame (0,0 1280x150)
        shows Header()
    Label (350,40 300x40), "COSMO"
    Label (120,150 150x30), "IPC Output"
    Label (320,150 150x30), "IPC Input"
    Label (340,200 170x30), "COSMO Standby"
    Lamp1 (300,205 20x20), variable: GVL.COSMO_Ready, style: Lamp-Lamp1-Red
    Label (340,230 170x30), "COSMO PASS"
    Lamp1 (300,235 20x20), variable: GVL.COSMO_OK, style: Lamp-Lamp1-Red
    Label (340,260 170x30), "COSMO FAIL"
    Lamp1 (300,265 20x20), variable: GVL.COSMO_NOTOK, style: Lamp-Lamp1-Red
    RoundedRectangle (110,200 150x40), "COSMO Run"
        toggle GVL.COSMO_Run
    Image (256,13 61x100), image: ImagePool.Icon-COSMO
    Image (677,141 269x439), image: ImagePool.Icon-COSMO
END_VISUALIZATION

// ---- VISUs/PAGE_JIG_C.TcVIS
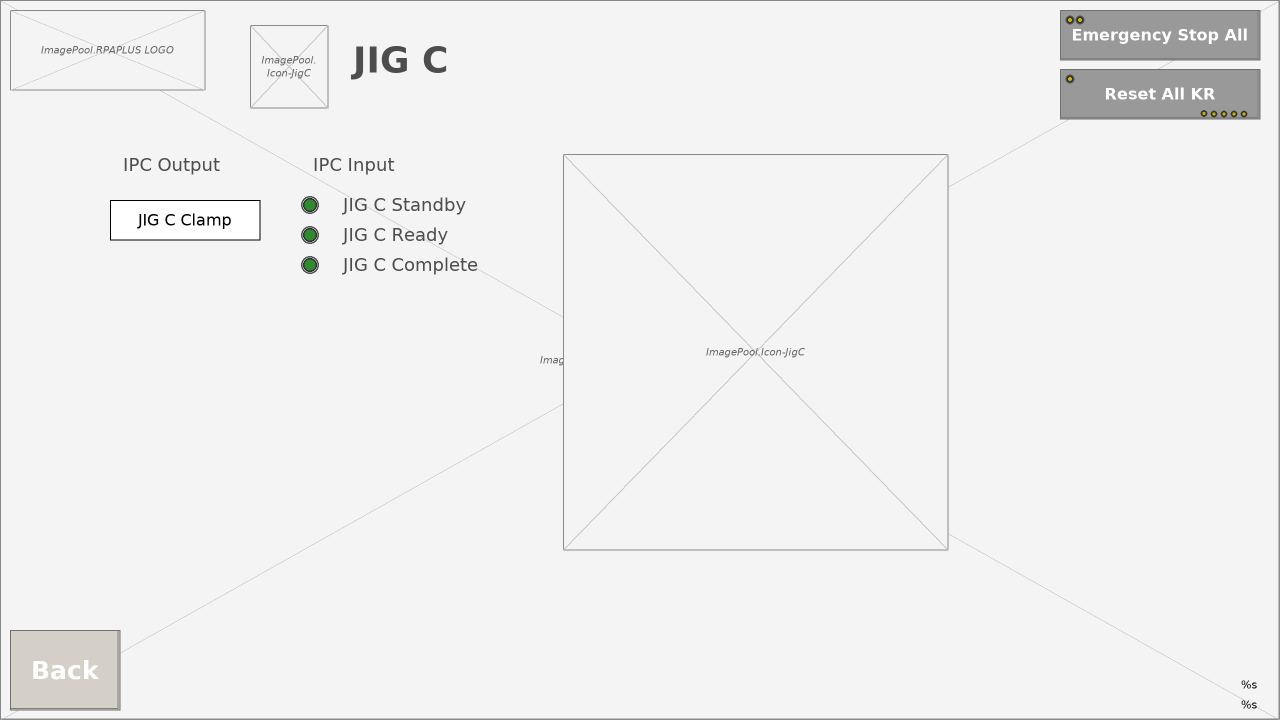
VISUALIZATION PAGE_JIG_C  // 1280x720
    Image (0,0 1280x720), image: ImagePool.The-New-Silver-Backgrounds
    Frame (0,620 1280x100)
        shows Footer_Back()
    Frame (0,0 1280x150)
        shows Header()
    Label (350,40 300x40), "JIG C"
    Label (120,150 150x30), "IPC Output"
    RoundedRectangle (110,200 150x40), "JIG C Clamp"
        toggle GVL.JIGC_Clamp
    Label (310,150 150x30), "IPC Input"
    Label (340,220 170x30), "JIG C Ready"
    Lamp1 (300,225 20x20), variable: GVL.JIGC_Ready, style: Lamp-Lamp1-Green
    Label (340,190 170x30), "JIG C Standby"
    Lamp1 (300,195 20x20), variable: GVL.JIGC_Standby, style: Lamp-Lamp1-Green
    Image (250,25 78x83), image: ImagePool.Icon-JigC
    Image (563,154 385x396), image: ImagePool.Icon-JigC
    Label (340,250 170x30), "JIG C Complete"
    Lamp1 (300,255 20x20), variable: GVL.JIGC_Complete, style: Lamp-Lamp1-Green
END_VISUALIZATION

// ---- VISUs/PAGE_CoolRack.TcVIS
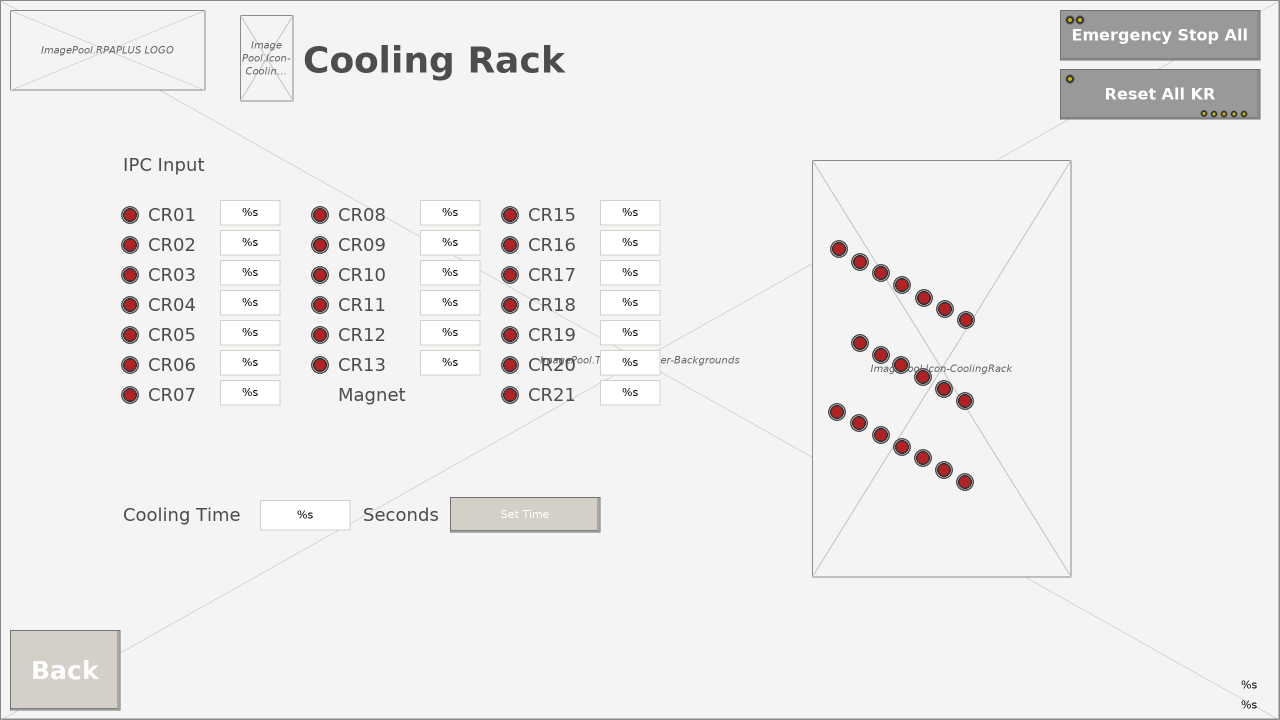
VISUALIZATION PAGE_CoolRack  // 1280x720
    Image (0,0 1280x720), image: ImagePool.The-New-Silver-Backgrounds
    Frame (0,620 1280x100)
        shows Footer_Back()
    Frame (0,0 1280x150)
        shows Header()
    Label (300,40 300x40), "Cooling Rack"
    Label (145,200 60x30), "CR01"
    Label (145,230 60x30), "CR02"
    Label (145,260 60x30), "CR03"
    Label (145,290 60x30), "CR04"
    Label (145,320 60x30), "CR05"
    Lamp1 (120,325 20x20), variable: COOL_RACK.CR[5], style: Lamp-Lamp1-Red
    Label (145,350 60x30), "CR06"
    Lamp1 (120,355 20x20), variable: COOL_RACK.CR[6], style: Lamp-Lamp1-Red
    Label (145,380 60x30), "CR07"
    Lamp1 (120,385 20x20), variable: COOL_RACK.CR[7], style: Lamp-Lamp1-Red
    Label (120,150 150x30), "IPC Input"
    Image (240,15 53x86), image: ImagePool.Icon-CoolingRack
    Image (812,160 259x417), image: ImagePool.Icon-CoolingRack
    Lamp1 (956,310 20x20), variable: COOL_RACK.CR[1], style: Lamp-Lamp1-Red
    Lamp1 (935,299 20x20), variable: COOL_RACK.CR[2], style: Lamp-Lamp1-Red
    Lamp1 (914,288 20x20), variable: COOL_RACK.CR[3], style: Lamp-Lamp1-Red
    Lamp1 (892,275 20x20), variable: COOL_RACK.CR[4], style: Lamp-Lamp1-Red
    Lamp1 (871,263 20x20), variable: COOL_RACK.CR[5], style: Lamp-Lamp1-Red
    Lamp1 (850,252 20x20), variable: COOL_RACK.CR[6], style: Lamp-Lamp1-Red
    Lamp1 (829,239 20x20), variable: COOL_RACK.CR[7], style: Lamp-Lamp1-Red
    Lamp1 (934,379 20x20), variable: COOL_RACK.CR[9], style: Lamp-Lamp1-Red
    Lamp1 (955,391 20x20), variable: COOL_RACK.CR[8], style: Lamp-Lamp1-Red
    Lamp1 (913,367 20x20), variable: COOL_RACK.CR[10], style: Lamp-Lamp1-Red
    Lamp1 (891,355 20x20), variable: COOL_RACK.CR[11], style: Lamp-Lamp1-Red
    Lamp1 (871,345 20x20), variable: COOL_RACK.CR[12], style: Lamp-Lamp1-Red
    Lamp1 (850,333 20x20), variable: COOL_RACK.CR[13], style: Lamp-Lamp1-Red
    Lamp1 (955,472 20x20), variable: COOL_RACK.CR[15], style: Lamp-Lamp1-Red
    Lamp1 (934,460 20x20), variable: COOL_RACK.CR[16], style: Lamp-Lamp1-Red
    Lamp1 (913,448 20x20), variable: COOL_RACK.CR[17], style: Lamp-Lamp1-Red
    Lamp1 (892,437 20x20), variable: COOL_RACK.CR[18], style: Lamp-Lamp1-Red
    Lamp1 (871,425 20x20), variable: COOL_RACK.CR[19], style: Lamp-Lamp1-Red
    Lamp1 (849,413 20x20), variable: COOL_RACK.CR[20], style: Lamp-Lamp1-Red
    Lamp1 (827,402 20x20), variable: COOL_RACK.CR[21], style: Lamp-Lamp1-Red
    Label (120,500 150x30), "Cooling Time"
    Textfield (260,500 90x30), "%s", text variable: GVL.iCooling_Time
        OnMouseClick: write the text variable via VisuDialogs.Numpad, min 1, max 1000, title 'Cooling Time (min)'
    Textfield (220,200 60x25), "%s", text variable: GVL.CRTimer[1]
    Textfield (220,230 60x25), "%s", text variable: GVL.CRTimer[2]
    Textfield (220,260 60x25), "%s", text variable: GVL.CRTimer[3]
    Textfield (220,290 60x25), "%s", text variable: GVL.CRTimer[4]
    Textfield (220,320 60x25), "%s", text variable: GVL.CRTimer[5]
    Textfield (220,350 60x25), "%s", text variable: GVL.CRTimer[6]
    Textfield (220,380 60x25), "%s", text variable: GVL.CRTimer[7]
    Label (335,200 60x30), "CR08"
    Lamp1 (310,205 20x20), variable: COOL_RACK.CR[8], style: Lamp-Lamp1-Red
    Label (335,230 60x30), "CR09"
    Lamp1 (310,235 20x20), variable: COOL_RACK.CR[9], style: Lamp-Lamp1-Red
    Label (335,260 60x30), "CR10"
    Lamp1 (310,265 20x20), variable: COOL_RACK.CR[10], style: Lamp-Lamp1-Red
    Label (335,290 60x30), "CR11"
    Lamp1 (310,295 20x20), variable: COOL_RACK.CR[11], style: Lamp-Lamp1-Red
    Label (335,320 60x30), "CR12"
    Lamp1 (310,325 20x20), variable: COOL_RACK.CR[12], style: Lamp-Lamp1-Red
    Label (335,350 60x30), "CR13"
    Lamp1 (310,355 20x20), variable: COOL_RACK.CR[13], style: Lamp-Lamp1-Red
    Label (335,380 91x30), "Magnet"
    Textfield (420,230 60x25), "%s", text variable: GVL.CRTimer[9]
    Textfield (420,200 60x25), "%s", text variable: GVL.CRTimer[8]
    Textfield (420,260 60x25), "%s", text variable: GVL.CRTimer[10]
    Textfield (420,290 60x25), "%s", text variable: GVL.CRTimer[11]
    Textfield (420,320 60x25), "%s", text variable: GVL.CRTimer[12]
    Textfield (420,350 60x25), "%s", text variable: GVL.CRTimer[13]
    Label (525,200 60x30), "CR15"
    Lamp1 (500,205 20x20), variable: COOL_RACK.CR[15], style: Lamp-Lamp1-Red
    Label (525,230 60x30), "CR16"
    Lamp1 (500,235 20x20), variable: COOL_RACK.CR[16], style: Lamp-Lamp1-Red
    Label (525,260 60x30), "CR17"
    Lamp1 (500,265 20x20), variable: COOL_RACK.CR[17], style: Lamp-Lamp1-Red
    Label (525,290 60x30), "CR18"
    Lamp1 (500,295 20x20), variable: COOL_RACK.CR[18], style: Lamp-Lamp1-Red
    Label (525,320 60x30), "CR19"
    Lamp1 (500,325 20x20), variable: COOL_RACK.CR[19], style: Lamp-Lamp1-Red
    Label (525,350 60x30), "CR20"
    Lamp1 (500,355 20x20), variable: COOL_RACK.CR[20], style: Lamp-Lamp1-Red
    Label (525,380 60x30), "CR21"
    Lamp1 (500,385 20x20), variable: COOL_RACK.CR[21], style: Lamp-Lamp1-Red
    Textfield (600,230 60x25), "%s", text variable: GVL.CRTimer[16]
    Textfield (600,200 60x25), "%s", text variable: GVL.CRTimer[15]
    Textfield (600,260 60x25), "%s", text variable: GVL.CRTimer[17]
    Textfield (600,290 60x25), "%s", text variable: GVL.CRTimer[18]
    Textfield (600,320 60x25), "%s", text variable: GVL.CRTimer[19]
    Textfield (600,350 60x25), "%s", text variable: GVL.CRTimer[20]
    Textfield (600,380 60x25), "%s", text variable: GVL.CRTimer[21]
    Button (450,497 150x35), "Set Time"
        tap COOL_RACK.set_time
    Label (360,500 80x30), "Seconds"
    Lamp1 (120,205 20x20), variable: COOL_RACK.CR[1], style: Lamp-Lamp1-Red
    Lamp1 (120,235 20x20), variable: COOL_RACK.CR[2], style: Lamp-Lamp1-Red
    Lamp1 (120,265 20x20), variable: COOL_RACK.CR[3], style: Lamp-Lamp1-Red
    Lamp1 (120,295 20x20), variable: COOL_RACK.CR[4], style: Lamp-Lamp1-Red
END_VISUALIZATION

// ---- VISUs/PAGE_JIG_A.TcVIS
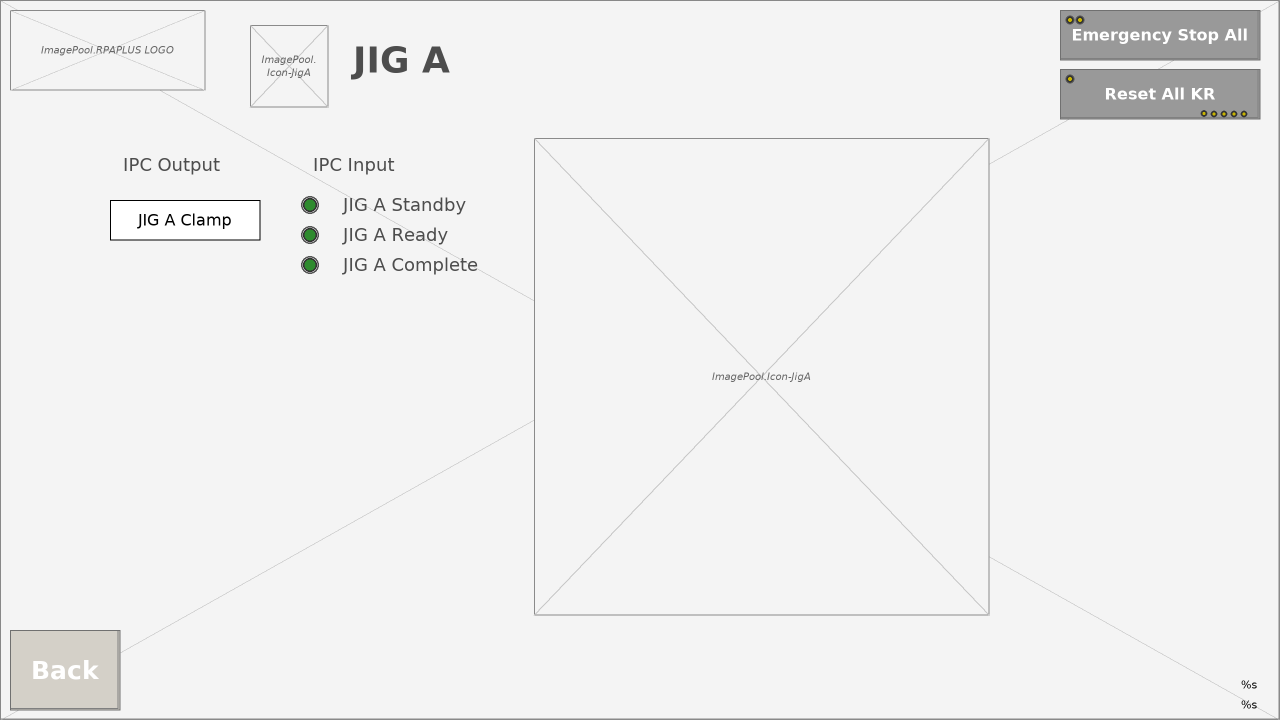
VISUALIZATION PAGE_JIG_A  // 1280x720
    Image (0,0 1280x720), image: ImagePool.The-New-Silver-Backgrounds
    Frame (0,620 1280x100)
        shows Footer_Back()
    Frame (0,0 1280x150)
        shows Header()
    Label (350,40 300x40), "JIG A"
    Label (120,150 150x30), "IPC Output"
    RoundedRectangle (110,200 150x40), "JIG A Clamp"
        toggle GVL.JIGA_Clamp
    Label (310,150 150x30), "IPC Input"
    Label (340,220 170x30), "JIG A Ready"
    Lamp1 (300,225 20x20), variable: GVL.JIGA_Ready, style: Lamp-Lamp1-Green
    Label (340,190 170x30), "JIG A Standby"
    Lamp1 (300,195 20x20), variable: GVL.JIGA_Standby, style: Lamp-Lamp1-Green
    Image (250,25 78x82), image: ImagePool.Icon-JigA
    Image (534,138 455x477), image: ImagePool.Icon-JigA
    Label (340,250 170x30), "JIG A Complete"
    Lamp1 (300,255 20x20), variable: GVL.JIGA_Complete, style: Lamp-Lamp1-Green
END_VISUALIZATION

// ---- VISUs/PAGE_JIG_B.TcVIS
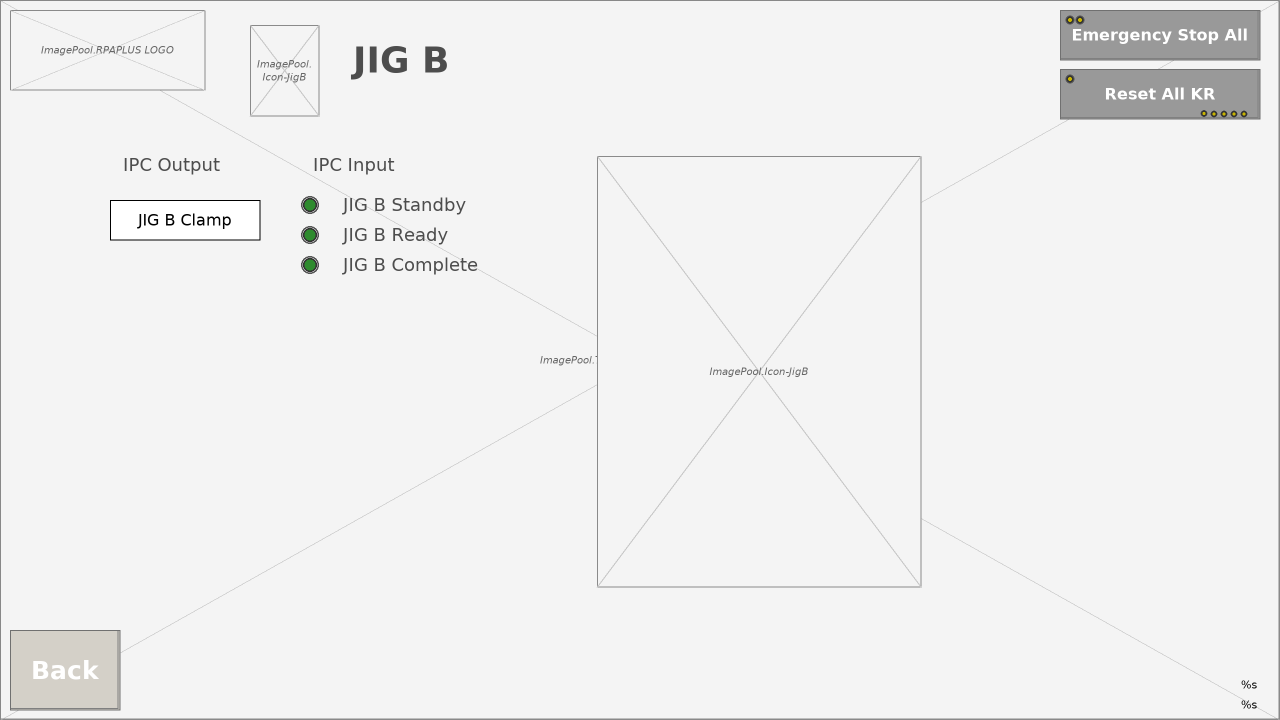
VISUALIZATION PAGE_JIG_B  // 1280x720
    Image (0,0 1280x720), image: ImagePool.The-New-Silver-Backgrounds
    Frame (0,620 1280x100)
        shows Footer_Back()
    Frame (0,0 1280x150)
        shows Header()
    Label (350,40 300x40), "JIG B"
    Label (120,150 150x30), "IPC Output"
    RoundedRectangle (110,200 150x40), "JIG B Clamp"
        toggle GVL.JIGB_Clamp
    Label (310,150 150x30), "IPC Input"
    Label (340,220 170x30), "JIG B Ready"
    Lamp1 (300,225 20x20), variable: GVL.JIGB_Ready, style: Lamp-Lamp1-Green
    Label (340,190 170x30), "JIG B Standby"
    Lamp1 (300,195 20x20), variable: GVL.JIGB_Standby, style: Lamp-Lamp1-Green
    Image (250,25 69x91), image: ImagePool.Icon-JigB
    Image (597,156 324x431), image: ImagePool.Icon-JigB
    Label (340,250 170x30), "JIG B Complete"
    Lamp1 (300,255 20x20), variable: GVL.JIGB_Complete, style: Lamp-Lamp1-Green
END_VISUALIZATION

// ---- VISUs/PAGE_KR1_Tab.TcVIS
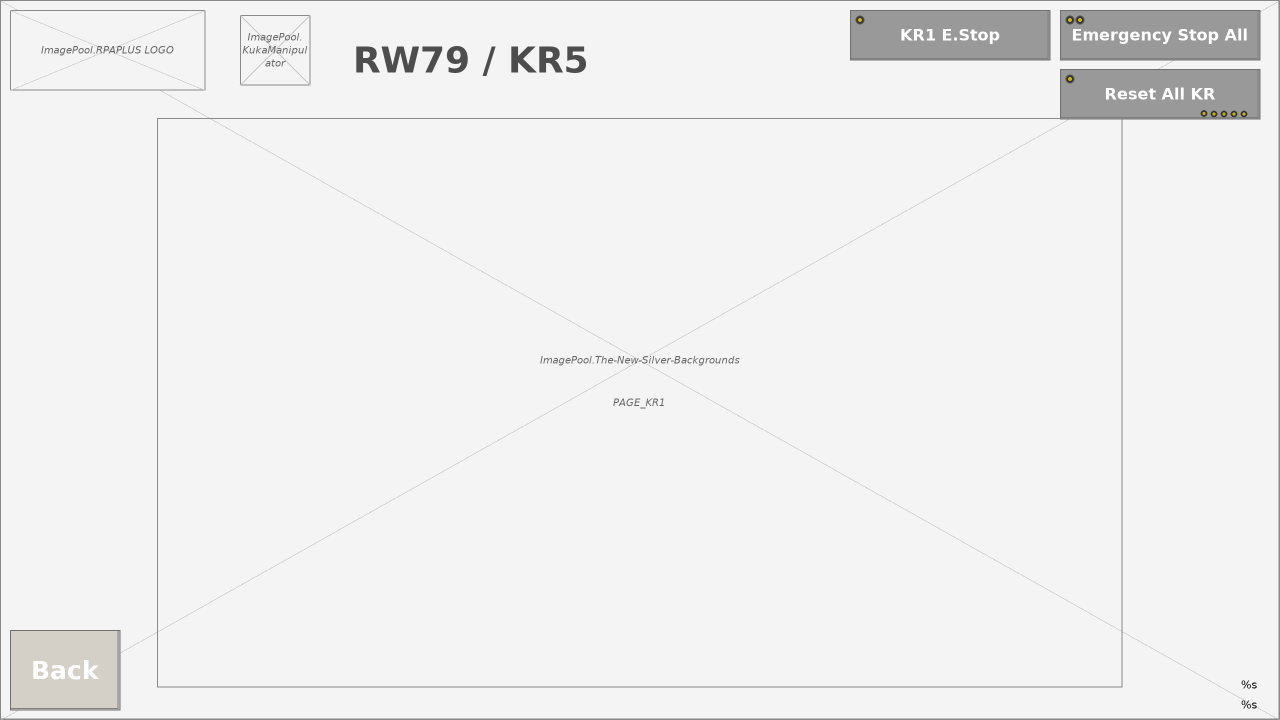
VISUALIZATION PAGE_KR1_Tab  // 1280x720
    Image (0,0 1280x720), image: ImagePool.The-New-Silver-Backgrounds
    Frame (0,620 1280x100)
        shows Footer_Back()
    Frame (0,0 1280x150)
        shows Header()
    Label (350,40 300x40), "RW79 / KR5"
    Group (850,10 200x50)
        Button (0,0 200x50), "KR1 E.Stop"
            toggle KR1.KR1_Estop
        Lamp1 (5,5 10x10), variable: KR1.KR1_Estop, style: Lamp-Lamp1-Yellow
    Image (240,15 70x70), image: ImagePool.KukaManipulator
    TabControl (157,118 965x569)
        shows PAGE_KR1()
        shows PAGE_KR1_Tab_1_100()
        shows PAGE_KR1_Tab_1_200()
        [0]: TabTitle=Main
        [1]: TabTitle=1-100
        [2]: TabTitle=100-200
END_VISUALIZATION

// ---- VISUs/PAGE_KR1_Tab_1_100.TcVIS
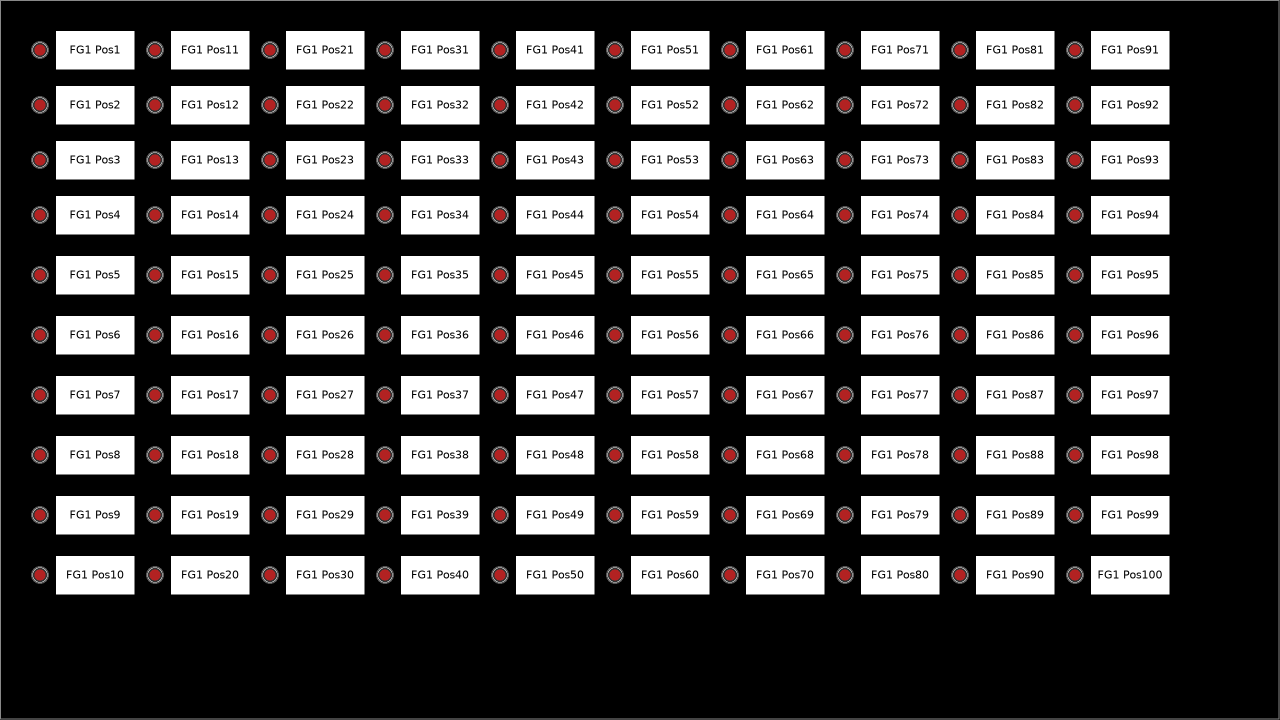
VISUALIZATION PAGE_KR1_Tab_1_100  // 1280x720
    RoundedRectangle (170,30 80x40), "FG1 Pos11"
        toggle KR1.bOutBit[5,4]
        OnMouseClick: execute {  }
    Lamp1 (145,40 20x20), variable: KR1.bInBit[5,4], style: Lamp-Lamp1-Red
    RoundedRectangle (55,30 80x40), "FG1 Pos1"
        toggle KR1.bOutBit[4,2]
        OnMouseClick: execute {  }
    Lamp1 (30,40 20x20), variable: KR1.bInBit[4,2], style: Lamp-Lamp1-Red
    RoundedRectangle (285,30 80x40), "FG1 Pos21"
        toggle KR1.bOutBit[6,6]
        OnMouseClick: execute {  }
    Lamp1 (260,40 20x20), variable: KR1.bInBit[6,6], style: Lamp-Lamp1-Red
    RoundedRectangle (400,30 80x40), "FG1 Pos31"
        toggle KR1.bOutBit[8,0]
        OnMouseClick: execute {  }
    Lamp1 (375,40 20x20), variable: KR1.bInBit[8,0], style: Lamp-Lamp1-Red
    RoundedRectangle (515,30 80x40), "FG1 Pos41"
        toggle KR1.bOutBit[9,2]
        OnMouseClick: execute {  }
    Lamp1 (490,40 20x20), variable: KR1.bInBit[9,2], style: Lamp-Lamp1-Red
    RoundedRectangle (745,30 80x40), "FG1 Pos61"
        toggle KR1.bOutBit[11,6]
        OnMouseClick: execute {  }
    Lamp1 (720,40 20x20), variable: KR1.bInBit[11,6], style: Lamp-Lamp1-Red
    RoundedRectangle (630,30 80x40), "FG1 Pos51"
        toggle KR1.bOutBit[10,4]
        OnMouseClick: execute {  }
    Lamp1 (605,40 20x20), variable: KR1.bInBit[10,4], style: Lamp-Lamp1-Red
    RoundedRectangle (860,30 80x40), "FG1 Pos71"
        toggle KR1.bOutBit[13,0]
        OnMouseClick: execute {  }
    Lamp1 (835,40 20x20), variable: KR1.bInBit[13,0], style: Lamp-Lamp1-Red
    RoundedRectangle (975,30 80x40), "FG1 Pos81"
        toggle KR1.bOutBit[14,2]
        OnMouseClick: execute {  }
    Lamp1 (950,40 20x20), variable: KR1.bInBit[14,2], style: Lamp-Lamp1-Red
    RoundedRectangle (1090,30 80x40), "FG1 Pos91"
        toggle KR1.bOutBit[15,4]
        OnMouseClick: execute {  }
    Lamp1 (1065,40 20x20), variable: KR1.bInBit[15,4], style: Lamp-Lamp1-Red
    RoundedRectangle (170,85 80x40), "FG1 Pos12"
        toggle KR1.bOutBit[5,5]
        OnMouseClick: execute {  }
    Lamp1 (145,95 20x20), variable: KR1.bInBit[5,5], style: Lamp-Lamp1-Red
    RoundedRectangle (55,85 80x40), "FG1 Pos2"
        toggle KR1.bOutBit[4,3]
        OnMouseClick: execute {  }
    Lamp1 (30,95 20x20), variable: KR1.bInBit[4,3], style: Lamp-Lamp1-Red
    RoundedRectangle (285,85 80x40), "FG1 Pos22"
        toggle KR1.bOutBit[6,7]
        OnMouseClick: execute {  }
    Lamp1 (260,95 20x20), variable: KR1.bInBit[6,7], style: Lamp-Lamp1-Red
    RoundedRectangle (400,85 80x40), "FG1 Pos32"
        toggle KR1.bOutBit[8,1]
        OnMouseClick: execute {  }
    Lamp1 (375,95 20x20), variable: KR1.bInBit[8,1], style: Lamp-Lamp1-Red
    RoundedRectangle (515,85 80x40), "FG1 Pos42"
        toggle KR1.bOutBit[9,3]
        OnMouseClick: execute {  }
    Lamp1 (490,95 20x20), variable: KR1.bInBit[9,3], style: Lamp-Lamp1-Red
    RoundedRectangle (745,85 80x40), "FG1 Pos62"
        toggle KR1.bOutBit[11,7]
        OnMouseClick: execute {  }
    Lamp1 (720,95 20x20), variable: KR1.bInBit[11,7], style: Lamp-Lamp1-Red
    RoundedRectangle (630,85 80x40), "FG1 Pos52"
        toggle KR1.bOutBit[10,5]
        OnMouseClick: execute {  }
    Lamp1 (605,95 20x20), variable: KR1.bInBit[10,5], style: Lamp-Lamp1-Red
    RoundedRectangle (860,85 80x40), "FG1 Pos72"
        toggle KR1.bOutBit[13,1]
        OnMouseClick: execute {  }
    Lamp1 (835,95 20x20), variable: KR1.bInBit[13,1], style: Lamp-Lamp1-Red
    RoundedRectangle (975,85 80x40), "FG1 Pos82"
        toggle KR1.bOutBit[14,3]
        OnMouseClick: execute {  }
    Lamp1 (950,95 20x20), variable: KR1.bInBit[14,3], style: Lamp-Lamp1-Red
    RoundedRectangle (1090,85 80x40), "FG1 Pos92"
        toggle KR1.bOutBit[15,5]
        OnMouseClick: execute {  }
    Lamp1 (1065,95 20x20), variable: KR1.bInBit[15,5], style: Lamp-Lamp1-Red
    RoundedRectangle (170,140 80x40), "FG1 Pos13"
        toggle KR1.bOutBit[5,6]
        OnMouseClick: execute {  }
    Lamp1 (145,150 20x20), variable: KR1.bInBit[5,6], style: Lamp-Lamp1-Red
    RoundedRectangle (55,140 80x40), "FG1 Pos3"
        toggle KR1.bOutBit[4,4]
        OnMouseClick: execute {  }
    Lamp1 (30,150 20x20), variable: KR1.bInBit[4,4], style: Lamp-Lamp1-Red
    RoundedRectangle (285,140 80x40), "FG1 Pos23"
        toggle KR1.bOutBit[7,0]
        OnMouseClick: execute {  }
    Lamp1 (260,150 20x20), variable: KR1.bInBit[7,0], style: Lamp-Lamp1-Red
    RoundedRectangle (400,140 80x40), "FG1 Pos33"
        toggle KR1.bOutBit[8,2]
        OnMouseClick: execute {  }
    Lamp1 (375,150 20x20), variable: KR1.bInBit[8,2], style: Lamp-Lamp1-Red
    RoundedRectangle (515,140 80x40), "FG1 Pos43"
        toggle KR1.bOutBit[9,4]
        OnMouseClick: execute {  }
    Lamp1 (490,150 20x20), variable: KR1.bInBit[9,4], style: Lamp-Lamp1-Red
    RoundedRectangle (745,140 80x40), "FG1 Pos63"
        toggle KR1.bOutBit[12,0]
        OnMouseClick: execute {  }
    Lamp1 (720,150 20x20), variable: KR1.bInBit[12,0], style: Lamp-Lamp1-Red
    RoundedRectangle (630,140 80x40), "FG1 Pos53"
        toggle KR1.bOutBit[10,6]
        OnMouseClick: execute {  }
    Lamp1 (605,150 20x20), variable: KR1.bInBit[10,6], style: Lamp-Lamp1-Red
    RoundedRectangle (860,140 80x40), "FG1 Pos73"
        toggle KR1.bOutBit[13,2]
        OnMouseClick: execute {  }
    Lamp1 (835,150 20x20), variable: KR1.bInBit[13,2], style: Lamp-Lamp1-Red
    RoundedRectangle (975,140 80x40), "FG1 Pos83"
        toggle KR1.bOutBit[14,4]
        OnMouseClick: execute {  }
    Lamp1 (950,150 20x20), variable: KR1.bInBit[14,4], style: Lamp-Lamp1-Red
    RoundedRectangle (1090,140 80x40), "FG1 Pos93"
        toggle KR1.bOutBit[15,6]
        OnMouseClick: execute {  }
    Lamp1 (1065,150 20x20), variable: KR1.bInBit[15,6], style: Lamp-Lamp1-Red
    RoundedRectangle (170,195 80x40), "FG1 Pos14"
        toggle KR1.bOutBit[5,7]
        OnMouseClick: execute {  }
    Lamp1 (145,205 20x20), variable: KR1.bInBit[5,7], style: Lamp-Lamp1-Red
    RoundedRectangle (55,195 80x40), "FG1 Pos4"
        toggle KR1.bOutBit[4,5]
        OnMouseClick: execute {  }
    Lamp1 (30,205 20x20), variable: KR1.bInBit[4,5], style: Lamp-Lamp1-Red
    RoundedRectangle (285,195 80x40), "FG1 Pos24"
        toggle KR1.bOutBit[7,1]
        OnMouseClick: execute {  }
    Lamp1 (260,205 20x20), variable: KR1.bInBit[7,1], style: Lamp-Lamp1-Red
    RoundedRectangle (400,195 80x40), "FG1 Pos34"
        toggle KR1.bOutBit[8,3]
        OnMouseClick: execute {  }
    Lamp1 (375,205 20x20), variable: KR1.bInBit[8,3], style: Lamp-Lamp1-Red
    RoundedRectangle (515,195 80x40), "FG1 Pos44"
        toggle KR1.bOutBit[9,5]
        OnMouseClick: execute {  }
    Lamp1 (490,205 20x20), variable: KR1.bInBit[9,5], style: Lamp-Lamp1-Red
    RoundedRectangle (745,195 80x40), "FG1 Pos64"
        toggle KR1.bOutBit[12,1]
        OnMouseClick: execute {  }
    Lamp1 (720,205 20x20), variable: KR1.bInBit[12,1], style: Lamp-Lamp1-Red
    RoundedRectangle (630,195 80x40), "FG1 Pos54"
        toggle KR1.bOutBit[10,7]
        OnMouseClick: execute {  }
    Lamp1 (605,205 20x20), variable: KR1.bInBit[10,7], style: Lamp-Lamp1-Red
    RoundedRectangle (860,195 80x40), "FG1 Pos74"
        toggle KR1.bOutBit[13,3]
        OnMouseClick: execute {  }
    Lamp1 (835,205 20x20), variable: KR1.bInBit[13,3], style: Lamp-Lamp1-Red
    RoundedRectangle (975,195 80x40), "FG1 Pos84"
        toggle KR1.bOutBit[14,5]
        OnMouseClick: execute {  }
    Lamp1 (950,205 20x20), variable: KR1.bInBit[14,5], style: Lamp-Lamp1-Red
    RoundedRectangle (1090,195 80x40), "FG1 Pos94"
        toggle KR1.bOutBit[15,7]
        OnMouseClick: execute {  }
    Lamp1 (1065,205 20x20), variable: KR1.bInBit[15,7], style: Lamp-Lamp1-Red
    RoundedRectangle (170,255 80x40), "FG1 Pos15"
        toggle KR1.bOutBit[6,0]
        OnMouseClick: execute {  }
    Lamp1 (145,265 20x20), variable: KR1.bInBit[6,0], style: Lamp-Lamp1-Red
    RoundedRectangle (55,255 80x40), "FG1 Pos5"
        toggle KR1.bOutBit[4,6]
        OnMouseClick: execute {  }
    Lamp1 (30,265 20x20), variable: KR1.bInBit[4,6], style: Lamp-Lamp1-Red
    RoundedRectangle (285,255 80x40), "FG1 Pos25"
        toggle KR1.bOutBit[7,2]
        OnMouseClick: execute {  }
    Lamp1 (260,265 20x20), variable: KR1.bInBit[7,2], style: Lamp-Lamp1-Red
    RoundedRectangle (400,255 80x40), "FG1 Pos35"
        toggle KR1.bOutBit[8,4]
        OnMouseClick: execute {  }
    Lamp1 (375,265 20x20), variable: KR1.bInBit[8,4], style: Lamp-Lamp1-Red
    RoundedRectangle (515,255 80x40), "FG1 Pos45"
        toggle KR1.bOutBit[9,6]
        OnMouseClick: execute {  }
    Lamp1 (490,265 20x20), variable: KR1.bInBit[9,6], style: Lamp-Lamp1-Red
    RoundedRectangle (745,255 80x40), "FG1 Pos65"
        toggle KR1.bOutBit[12,2]
        OnMouseClick: execute {  }
    Lamp1 (720,265 20x20), variable: KR1.bInBit[12,2], style: Lamp-Lamp1-Red
    RoundedRectangle (630,255 80x40), "FG1 Pos55"
        toggle KR1.bOutBit[11,0]
        OnMouseClick: execute {  }
    Lamp1 (605,265 20x20), variable: KR1.bInBit[11,0], style: Lamp-Lamp1-Red
    RoundedRectangle (860,255 80x40), "FG1 Pos75"
        toggle KR1.bOutBit[13,4]
        OnMouseClick: execute {  }
    Lamp1 (835,265 20x20), variable: KR1.bInBit[13,4], style: Lamp-Lamp1-Red
    RoundedRectangle (975,255 80x40), "FG1 Pos85"
        toggle KR1.bOutBit[14,6]
        OnMouseClick: execute {  }
    Lamp1 (950,265 20x20), variable: KR1.bInBit[14,6], style: Lamp-Lamp1-Red
    RoundedRectangle (1090,255 80x40), "FG1 Pos95"
        toggle KR1.bOutBit[16,0]
        OnMouseClick: execute {  }
    Lamp1 (1065,265 20x20), variable: KR1.bInBit[16,0], style: Lamp-Lamp1-Red
    RoundedRectangle (170,315 80x40), "FG1 Pos16"
        toggle KR1.bOutBit[6,1]
        OnMouseClick: execute {  }
    Lamp1 (145,325 20x20), variable: KR1.bInBit[6,1], style: Lamp-Lamp1-Red
    RoundedRectangle (55,315 80x40), "FG1 Pos6"
        toggle KR1.bOutBit[4,7]
        OnMouseClick: execute {  }
    Lamp1 (30,325 20x20), variable: KR1.bInBit[4,7], style: Lamp-Lamp1-Red
    RoundedRectangle (285,315 80x40), "FG1 Pos26"
        toggle KR1.bOutBit[7,3]
        OnMouseClick: execute {  }
    Lamp1 (260,325 20x20), variable: KR1.bInBit[7,3], style: Lamp-Lamp1-Red
    RoundedRectangle (400,315 80x40), "FG1 Pos36"
        toggle KR1.bOutBit[8,5]
        OnMouseClick: execute {  }
    Lamp1 (375,325 20x20), variable: KR1.bInBit[8,5], style: Lamp-Lamp1-Red
    RoundedRectangle (515,315 80x40), "FG1 Pos46"
        toggle KR1.bOutBit[9,7]
        OnMouseClick: execute {  }
    Lamp1 (490,325 20x20), variable: KR1.bInBit[9,7], style: Lamp-Lamp1-Red
    RoundedRectangle (745,315 80x40), "FG1 Pos66"
        toggle KR1.bOutBit[12,3]
        OnMouseClick: execute {  }
    Lamp1 (720,325 20x20), variable: KR1.bInBit[12,3], style: Lamp-Lamp1-Red
    RoundedRectangle (630,315 80x40), "FG1 Pos56"
        toggle KR1.bOutBit[11,1]
        OnMouseClick: execute {  }
    Lamp1 (605,325 20x20), variable: KR1.bInBit[11,1], style: Lamp-Lamp1-Red
    RoundedRectangle (860,315 80x40), "FG1 Pos76"
        toggle KR1.bOutBit[13,5]
        OnMouseClick: execute {  }
    Lamp1 (835,325 20x20), variable: KR1.bInBit[13,5], style: Lamp-Lamp1-Red
    RoundedRectangle (975,315 80x40), "FG1 Pos86"
        toggle KR1.bOutBit[14,7]
        OnMouseClick: execute {  }
    Lamp1 (950,325 20x20), variable: KR1.bInBit[14,7], style: Lamp-Lamp1-Red
    RoundedRectangle (1090,315 80x40), "FG1 Pos96"
        toggle KR1.bOutBit[16,1]
        OnMouseClick: execute {  }
    Lamp1 (1065,325 20x20), variable: KR1.bInBit[16,1], style: Lamp-Lamp1-Red
    RoundedRectangle (170,375 80x40), "FG1 Pos17"
        toggle KR1.bOutBit[6,2]
        OnMouseClick: execute {  }
    Lamp1 (145,385 20x20), variable: KR1.bInBit[6,2], style: Lamp-Lamp1-Red
    RoundedRectangle (55,375 80x40), "FG1 Pos7"
        toggle KR1.bOutBit[5,0]
        OnMouseClick: execute {  }
    Lamp1 (30,385 20x20), variable: KR1.bInBit[5,0], style: Lamp-Lamp1-Red
    RoundedRectangle (285,375 80x40), "FG1 Pos27"
        toggle KR1.bOutBit[7,4]
        OnMouseClick: execute {  }
    Lamp1 (260,385 20x20), variable: KR1.bInBit[7,4], style: Lamp-Lamp1-Red
    RoundedRectangle (400,375 80x40), "FG1 Pos37"
        toggle KR1.bOutBit[8,6]
        OnMouseClick: execute {  }
    Lamp1 (375,385 20x20), variable: KR1.bInBit[8,6], style: Lamp-Lamp1-Red
    RoundedRectangle (515,375 80x40), "FG1 Pos47"
        toggle KR1.bOutBit[10,0]
        OnMouseClick: execute {  }
    Lamp1 (490,385 20x20), variable: KR1.bInBit[10,0], style: Lamp-Lamp1-Red
    RoundedRectangle (745,375 80x40), "FG1 Pos67"
        toggle KR1.bOutBit[12,4]
        OnMouseClick: execute {  }
    Lamp1 (720,385 20x20), variable: KR1.bInBit[12,4], style: Lamp-Lamp1-Red
    RoundedRectangle (630,375 80x40), "FG1 Pos57"
        toggle KR1.bOutBit[11,2]
        OnMouseClick: execute {  }
    Lamp1 (605,385 20x20), variable: KR1.bInBit[11,2], style: Lamp-Lamp1-Red
    RoundedRectangle (860,375 80x40), "FG1 Pos77"
        toggle KR1.bOutBit[13,6]
        OnMouseClick: execute {  }
    Lamp1 (835,385 20x20), variable: KR1.bInBit[13,6], style: Lamp-Lamp1-Red
    RoundedRectangle (975,375 80x40), "FG1 Pos87"
        toggle KR1.bOutBit[15,0]
        OnMouseClick: execute {  }
    Lamp1 (950,385 20x20), variable: KR1.bInBit[15,0], style: Lamp-Lamp1-Red
    RoundedRectangle (1090,375 80x40), "FG1 Pos97"
        toggle KR1.bOutBit[16,2]
        OnMouseClick: execute {  }
    Lamp1 (1065,385 20x20), variable: KR1.bInBit[16,2], style: Lamp-Lamp1-Red
    RoundedRectangle (170,435 80x40), "FG1 Pos18"
        toggle KR1.bOutBit[6,3]
        OnMouseClick: execute {  }
    Lamp1 (145,445 20x20), variable: KR1.bInBit[6,3], style: Lamp-Lamp1-Red
    RoundedRectangle (55,435 80x40), "FG1 Pos8"
        toggle KR1.bOutBit[5,1]
        OnMouseClick: execute {  }
    Lamp1 (30,445 20x20), variable: KR1.bInBit[5,1], style: Lamp-Lamp1-Red
    RoundedRectangle (285,435 80x40), "FG1 Pos28"
        toggle KR1.bOutBit[7,5]
        OnMouseClick: execute {  }
    Lamp1 (260,445 20x20), variable: KR1.bInBit[7,5], style: Lamp-Lamp1-Red
    RoundedRectangle (400,435 80x40), "FG1 Pos38"
        toggle KR1.bOutBit[8,7]
        OnMouseClick: execute {  }
    Lamp1 (375,445 20x20), variable: KR1.bInBit[8,7], style: Lamp-Lamp1-Red
    RoundedRectangle (515,435 80x40), "FG1 Pos48"
        toggle KR1.bOutBit[10,1]
        OnMouseClick: execute {  }
    Lamp1 (490,445 20x20), variable: KR1.bInBit[10,1], style: Lamp-Lamp1-Red
    RoundedRectangle (745,435 80x40), "FG1 Pos68"
        toggle KR1.bOutBit[12,5]
        OnMouseClick: execute {  }
    Lamp1 (720,445 20x20), variable: KR1.bInBit[12,5], style: Lamp-Lamp1-Red
    RoundedRectangle (630,435 80x40), "FG1 Pos58"
        toggle KR1.bOutBit[11,3]
        OnMouseClick: execute {  }
    Lamp1 (605,445 20x20), variable: KR1.bInBit[11,3], style: Lamp-Lamp1-Red
    RoundedRectangle (860,435 80x40), "FG1 Pos78"
        toggle KR1.bOutBit[13,7]
        OnMouseClick: execute {  }
    Lamp1 (835,445 20x20), variable: KR1.bInBit[13,7], style: Lamp-Lamp1-Red
    RoundedRectangle (975,435 80x40), "FG1 Pos88"
        toggle KR1.bOutBit[15,1]
        OnMouseClick: execute {  }
    Lamp1 (950,445 20x20), variable: KR1.bInBit[15,1], style: Lamp-Lamp1-Red
    RoundedRectangle (1090,435 80x40), "FG1 Pos98"
        toggle KR1.bOutBit[16,3]
        OnMouseClick: execute {  }
    Lamp1 (1065,445 20x20), variable: KR1.bInBit[16,3], style: Lamp-Lamp1-Red
    RoundedRectangle (55,495 80x40), "FG1 Pos9"
        toggle KR1.bOutBit[5,2]
        OnMouseClick: execute {  }
    Lamp1 (30,505 20x20), variable: KR1.bInBit[5,2], style: Lamp-Lamp1-Red
    RoundedRectangle (170,495 80x40), "FG1 Pos19"
        toggle KR1.bOutBit[6,4]
        OnMouseClick: execute {  }
    Lamp1 (145,505 20x20), variable: KR1.bInBit[6,4], style: Lamp-Lamp1-Red
    RoundedRectangle (285,495 80x40), "FG1 Pos29"
        toggle KR1.bOutBit[7,6]
        OnMouseClick: execute {  }
    Lamp1 (260,505 20x20), variable: KR1.bInBit[7,6], style: Lamp-Lamp1-Red
    RoundedRectangle (400,495 80x40), "FG1 Pos39"
        toggle KR1.bOutBit[9,0]
        OnMouseClick: execute {  }
    Lamp1 (375,505 20x20), variable: KR1.bInBit[9,0], style: Lamp-Lamp1-Red
    RoundedRectangle (515,495 80x40), "FG1 Pos49"
        toggle KR1.bOutBit[10,2]
        OnMouseClick: execute {  }
    Lamp1 (490,505 20x20), variable: KR1.bInBit[10,2], style: Lamp-Lamp1-Red
    RoundedRectangle (630,495 80x40), "FG1 Pos59"
        toggle KR1.bOutBit[11,4]
        OnMouseClick: execute {  }
    Lamp1 (605,505 20x20), variable: KR1.bInBit[11,4], style: Lamp-Lamp1-Red
    RoundedRectangle (745,495 80x40), "FG1 Pos69"
        toggle KR1.bOutBit[12,6]
        OnMouseClick: execute {  }
    Lamp1 (720,505 20x20), variable: KR1.bInBit[12,6], style: Lamp-Lamp1-Red
    RoundedRectangle (860,495 80x40), "FG1 Pos79"
        toggle KR1.bOutBit[14,0]
        OnMouseClick: execute {  }
    Lamp1 (835,505 20x20), variable: KR1.bInBit[14,0], style: Lamp-Lamp1-Red
    RoundedRectangle (975,495 80x40), "FG1 Pos89"
        toggle KR1.bOutBit[15,2]
        OnMouseClick: execute {  }
    Lamp1 (950,505 20x20), variable: KR1.bInBit[15,2], style: Lamp-Lamp1-Red
    RoundedRectangle (1090,495 80x40), "FG1 Pos99"
        toggle KR1.bOutBit[16,4]
        OnMouseClick: execute {  }
    Lamp1 (1065,505 20x20), variable: KR1.bInBit[16,4], style: Lamp-Lamp1-Red
    RoundedRectangle (55,555 80x40), "FG1 Pos10"
        toggle KR1.bOutBit[5,3]
        OnMouseClick: execute {  }
    Lamp1 (30,565 20x20), variable: KR1.bInBit[5,3], style: Lamp-Lamp1-Red
    RoundedRectangle (170,555 80x40), "FG1 Pos20"
        toggle KR1.bOutBit[6,5]
        OnMouseClick: execute {  }
    Lamp1 (145,565 20x20), variable: KR1.bInBit[6,5], style: Lamp-Lamp1-Red
    RoundedRectangle (285,555 80x40), "FG1 Pos30"
        toggle KR1.bOutBit[7,7]
        OnMouseClick: execute {  }
    Lamp1 (260,565 20x20), variable: KR1.bInBit[7,7], style: Lamp-Lamp1-Red
    RoundedRectangle (400,555 80x40), "FG1 Pos40"
        toggle KR1.bOutBit[9,1]
        OnMouseClick: execute {  }
    Lamp1 (375,565 20x20), variable: KR1.bInBit[9,1], style: Lamp-Lamp1-Red
    RoundedRectangle (515,555 80x40), "FG1 Pos50"
        toggle KR1.bOutBit[10,3]
        OnMouseClick: execute {  }
    Lamp1 (490,565 20x20), variable: KR1.bInBit[10,3], style: Lamp-Lamp1-Red
    RoundedRectangle (630,555 80x40), "FG1 Pos60"
        toggle KR1.bOutBit[11,5]
        OnMouseClick: execute {  }
    Lamp1 (605,565 20x20), variable: KR1.bInBit[11,5], style: Lamp-Lamp1-Red
    RoundedRectangle (745,555 80x40), "FG1 Pos70"
        toggle KR1.bOutBit[12,7]
        OnMouseClick: execute {  }
    Lamp1 (720,565 20x20), variable: KR1.bInBit[12,7], style: Lamp-Lamp1-Red
    RoundedRectangle (860,555 80x40), "FG1 Pos80"
        toggle KR1.bOutBit[14,1]
        OnMouseClick: execute {  }
    Lamp1 (835,565 20x20), variable: KR1.bInBit[14,1], style: Lamp-Lamp1-Red
    RoundedRectangle (975,555 80x40), "FG1 Pos90"
        toggle KR1.bOutBit[15,3]
        OnMouseClick: execute {  }
    Lamp1 (950,565 20x20), variable: KR1.bInBit[15,3], style: Lamp-Lamp1-Red
    RoundedRectangle (1090,555 80x40), "FG1 Pos100"
        toggle KR1.bOutBit[16,5]
        OnMouseClick: execute {  }
    Lamp1 (1065,565 20x20), variable: KR1.bInBit[16,5], style: Lamp-Lamp1-Red
END_VISUALIZATION

// ---- VISUs/PAGE_KR1_Tab_1_200.TcVIS
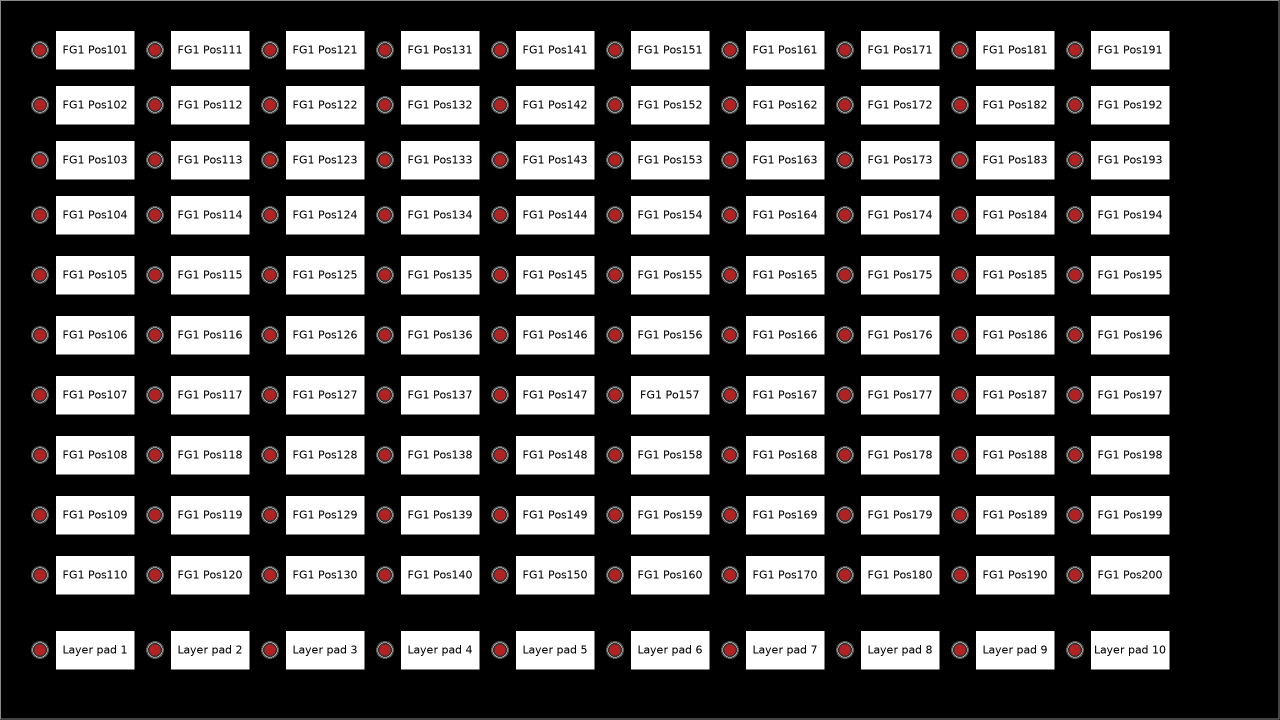
VISUALIZATION PAGE_KR1_Tab_1_200  // 1280x720
    RoundedRectangle (170,30 80x40), "FG1 Pos111"
        toggle KR1.bOutBit[18,0]
        OnMouseClick: execute {  }
    Lamp1 (145,40 20x20), variable: KR1.bInBit[18,0], style: Lamp-Lamp1-Red
    RoundedRectangle (55,30 80x40), "FG1 Pos101"
        toggle KR1.bOutBit[16,6]
        OnMouseClick: execute {  }
    Lamp1 (30,40 20x20), variable: KR1.bInBit[16,6], style: Lamp-Lamp1-Red
    RoundedRectangle (285,30 80x40), "FG1 Pos121"
        toggle KR1.bOutBit[19,2]
        OnMouseClick: execute {  }
    Lamp1 (260,40 20x20), variable: KR1.bInBit[19,2], style: Lamp-Lamp1-Red
    RoundedRectangle (400,30 80x40), "FG1 Pos131"
        toggle KR1.bOutBit[20,4]
        OnMouseClick: execute {  }
    Lamp1 (375,40 20x20), variable: KR1.bInBit[20,4], style: Lamp-Lamp1-Red
    RoundedRectangle (515,30 80x40), "FG1 Pos141"
        toggle KR1.bOutBit[21,6]
        OnMouseClick: execute {  }
    Lamp1 (490,40 20x20), variable: KR1.bInBit[21,6], style: Lamp-Lamp1-Red
    RoundedRectangle (745,30 80x40), "FG1 Pos161"
        toggle KR1.bOutBit[24,2]
        OnMouseClick: execute {  }
    Lamp1 (720,40 20x20), variable: KR1.bInBit[24,2], style: Lamp-Lamp1-Red
    RoundedRectangle (630,30 80x40), "FG1 Pos151"
        toggle KR1.bOutBit[23,0]
        OnMouseClick: execute {  }
    Lamp1 (605,40 20x20), variable: KR1.bInBit[23,0], style: Lamp-Lamp1-Red
    RoundedRectangle (860,30 80x40), "FG1 Pos171"
        toggle KR1.bOutBit[25,4]
        OnMouseClick: execute {  }
    Lamp1 (835,40 20x20), variable: KR1.bInBit[25,4], style: Lamp-Lamp1-Red
    RoundedRectangle (975,30 80x40), "FG1 Pos181"
        toggle KR1.bOutBit[26,6]
        OnMouseClick: execute {  }
    Lamp1 (950,40 20x20), variable: KR1.bInBit[26,6], style: Lamp-Lamp1-Red
    RoundedRectangle (1090,30 80x40), "FG1 Pos191"
        toggle KR1.bOutBit[28,0]
        OnMouseClick: execute {  }
    Lamp1 (1065,40 20x20), variable: KR1.bInBit[28,0], style: Lamp-Lamp1-Red
    RoundedRectangle (170,85 80x40), "FG1 Pos112"
        toggle KR1.bOutBit[18,1]
        OnMouseClick: execute {  }
    Lamp1 (145,95 20x20), variable: KR1.bInBit[18,1], style: Lamp-Lamp1-Red
    RoundedRectangle (55,85 80x40), "FG1 Pos102"
        toggle KR1.bOutBit[16,7]
        OnMouseClick: execute {  }
    Lamp1 (30,95 20x20), variable: KR1.bInBit[16,7], style: Lamp-Lamp1-Red
    RoundedRectangle (285,85 80x40), "FG1 Pos122"
        toggle KR1.bOutBit[19,3]
        OnMouseClick: execute {  }
    Lamp1 (260,95 20x20), variable: KR1.bInBit[19,3], style: Lamp-Lamp1-Red
    RoundedRectangle (400,85 80x40), "FG1 Pos132"
        toggle KR1.bOutBit[20,5]
        OnMouseClick: execute {  }
    Lamp1 (375,95 20x20), variable: KR1.bInBit[20,5], style: Lamp-Lamp1-Red
    RoundedRectangle (515,85 80x40), "FG1 Pos142"
        toggle KR1.bOutBit[21,7]
        OnMouseClick: execute {  }
    Lamp1 (490,95 20x20), variable: KR1.bInBit[21,7], style: Lamp-Lamp1-Red
    RoundedRectangle (745,85 80x40), "FG1 Pos162"
        toggle KR1.bOutBit[24,3]
        OnMouseClick: execute {  }
    Lamp1 (720,95 20x20), variable: KR1.bInBit[24,3], style: Lamp-Lamp1-Red
    RoundedRectangle (630,85 80x40), "FG1 Pos152"
        toggle KR1.bOutBit[23,1]
        OnMouseClick: execute {  }
    Lamp1 (605,95 20x20), variable: KR1.bInBit[23,1], style: Lamp-Lamp1-Red
    RoundedRectangle (860,85 80x40), "FG1 Pos172"
        toggle KR1.bOutBit[25,5]
        OnMouseClick: execute {  }
    Lamp1 (835,95 20x20), variable: KR1.bInBit[25,5], style: Lamp-Lamp1-Red
    RoundedRectangle (975,85 80x40), "FG1 Pos182"
        toggle KR1.bOutBit[26,7]
        OnMouseClick: execute {  }
    Lamp1 (950,95 20x20), variable: KR1.bInBit[26,7], style: Lamp-Lamp1-Red
    RoundedRectangle (1090,85 80x40), "FG1 Pos192"
        toggle KR1.bOutBit[28,1]
        OnMouseClick: execute {  }
    Lamp1 (1065,95 20x20), variable: KR1.bInBit[28,1], style: Lamp-Lamp1-Red
    RoundedRectangle (170,140 80x40), "FG1 Pos113"
        toggle KR1.bOutBit[18,2]
        OnMouseClick: execute {  }
    Lamp1 (145,150 20x20), variable: KR1.bInBit[18,2], style: Lamp-Lamp1-Red
    RoundedRectangle (55,140 80x40), "FG1 Pos103"
        toggle KR1.bOutBit[17,0]
        OnMouseClick: execute {  }
    Lamp1 (30,150 20x20), variable: KR1.bInBit[17,0], style: Lamp-Lamp1-Red
    RoundedRectangle (285,140 80x40), "FG1 Pos123"
        toggle KR1.bOutBit[19,4]
        OnMouseClick: execute {  }
    Lamp1 (260,150 20x20), variable: KR1.bInBit[19,4], style: Lamp-Lamp1-Red
    RoundedRectangle (400,140 80x40), "FG1 Pos133"
        toggle KR1.bOutBit[20,6]
        OnMouseClick: execute {  }
    Lamp1 (375,150 20x20), variable: KR1.bInBit[20,6], style: Lamp-Lamp1-Red
    RoundedRectangle (515,140 80x40), "FG1 Pos143"
        toggle KR1.bOutBit[22,0]
        OnMouseClick: execute {  }
    Lamp1 (490,150 20x20), variable: KR1.bInBit[22,0], style: Lamp-Lamp1-Red
    RoundedRectangle (745,140 80x40), "FG1 Pos163"
        toggle KR1.bOutBit[24,4]
        OnMouseClick: execute {  }
    Lamp1 (720,150 20x20), variable: KR1.bInBit[24,4], style: Lamp-Lamp1-Red
    RoundedRectangle (630,140 80x40), "FG1 Pos153"
        toggle KR1.bOutBit[23,2]
        OnMouseClick: execute {  }
    Lamp1 (605,150 20x20), variable: KR1.bInBit[23,2], style: Lamp-Lamp1-Red
    RoundedRectangle (860,140 80x40), "FG1 Pos173"
        toggle KR1.bOutBit[25,6]
        OnMouseClick: execute {  }
    Lamp1 (835,150 20x20), variable: KR1.bInBit[25,6], style: Lamp-Lamp1-Red
    RoundedRectangle (975,140 80x40), "FG1 Pos183"
        toggle KR1.bOutBit[27,0]
        OnMouseClick: execute {  }
    Lamp1 (950,150 20x20), variable: KR1.bInBit[27,0], style: Lamp-Lamp1-Red
    RoundedRectangle (1090,140 80x40), "FG1 Pos193"
        toggle KR1.bOutBit[28,2]
        OnMouseClick: execute {  }
    Lamp1 (1065,150 20x20), variable: KR1.bInBit[28,2], style: Lamp-Lamp1-Red
    RoundedRectangle (170,195 80x40), "FG1 Pos114"
        toggle KR1.bOutBit[18,3]
        OnMouseClick: execute {  }
    Lamp1 (145,205 20x20), variable: KR1.bInBit[18,3], style: Lamp-Lamp1-Red
    RoundedRectangle (55,195 80x40), "FG1 Pos104"
        toggle KR1.bOutBit[17,1]
        OnMouseClick: execute {  }
    Lamp1 (30,205 20x20), variable: KR1.bInBit[17,1], style: Lamp-Lamp1-Red
    RoundedRectangle (285,195 80x40), "FG1 Pos124"
        toggle KR1.bOutBit[19,5]
        OnMouseClick: execute {  }
    Lamp1 (260,205 20x20), variable: KR1.bInBit[19,5], style: Lamp-Lamp1-Red
    RoundedRectangle (400,195 80x40), "FG1 Pos134"
        toggle KR1.bOutBit[20,7]
        OnMouseClick: execute {  }
    Lamp1 (375,205 20x20), variable: KR1.bInBit[20,7], style: Lamp-Lamp1-Red
    RoundedRectangle (515,195 80x40), "FG1 Pos144"
        toggle KR1.bOutBit[22,1]
        OnMouseClick: execute {  }
    Lamp1 (490,205 20x20), variable: KR1.bInBit[22,1], style: Lamp-Lamp1-Red
    RoundedRectangle (745,195 80x40), "FG1 Pos164"
        toggle KR1.bOutBit[24,5]
        OnMouseClick: execute {  }
    Lamp1 (720,205 20x20), variable: KR1.bInBit[24,5], style: Lamp-Lamp1-Red
    RoundedRectangle (630,195 80x40), "FG1 Pos154"
        toggle KR1.bOutBit[23,3]
        OnMouseClick: execute {  }
    Lamp1 (605,205 20x20), variable: KR1.bInBit[23,3], style: Lamp-Lamp1-Red
    RoundedRectangle (860,195 80x40), "FG1 Pos174"
        toggle KR1.bOutBit[25,7]
        OnMouseClick: execute {  }
    Lamp1 (835,205 20x20), variable: KR1.bInBit[25,7], style: Lamp-Lamp1-Red
    RoundedRectangle (975,195 80x40), "FG1 Pos184"
        toggle KR1.bOutBit[27,1]
        OnMouseClick: execute {  }
    Lamp1 (950,205 20x20), variable: KR1.bInBit[27,1], style: Lamp-Lamp1-Red
    RoundedRectangle (1090,195 80x40), "FG1 Pos194"
        toggle KR1.bOutBit[28,3]
        OnMouseClick: execute {  }
    Lamp1 (1065,205 20x20), variable: KR1.bInBit[28,3], style: Lamp-Lamp1-Red
    RoundedRectangle (170,255 80x40), "FG1 Pos115"
        toggle KR1.bOutBit[18,4]
        OnMouseClick: execute {  }
    Lamp1 (145,265 20x20), variable: KR1.bInBit[18,4], style: Lamp-Lamp1-Red
    RoundedRectangle (55,255 80x40), "FG1 Pos105"
        toggle KR1.bOutBit[17,2]
        OnMouseClick: execute {  }
    Lamp1 (30,265 20x20), variable: KR1.bInBit[17,2], style: Lamp-Lamp1-Red
    RoundedRectangle (285,255 80x40), "FG1 Pos125"
        toggle KR1.bOutBit[19,6]
        OnMouseClick: execute {  }
    Lamp1 (260,265 20x20), variable: KR1.bInBit[19,6], style: Lamp-Lamp1-Red
    RoundedRectangle (400,255 80x40), "FG1 Pos135"
        toggle KR1.bOutBit[21,0]
        OnMouseClick: execute {  }
    Lamp1 (375,265 20x20), variable: KR1.bInBit[21,0], style: Lamp-Lamp1-Red
    RoundedRectangle (515,255 80x40), "FG1 Pos145"
        toggle KR1.bOutBit[22,2]
        OnMouseClick: execute {  }
    Lamp1 (490,265 20x20), variable: KR1.bInBit[22,2], style: Lamp-Lamp1-Red
    RoundedRectangle (745,255 80x40), "FG1 Pos165"
        toggle KR1.bOutBit[24,6]
        OnMouseClick: execute {  }
    Lamp1 (720,265 20x20), variable: KR1.bInBit[24,6], style: Lamp-Lamp1-Red
    RoundedRectangle (630,255 80x40), "FG1 Pos155"
        toggle KR1.bOutBit[23,4]
        OnMouseClick: execute {  }
    Lamp1 (605,265 20x20), variable: KR1.bInBit[23,4], style: Lamp-Lamp1-Red
    RoundedRectangle (860,255 80x40), "FG1 Pos175"
        toggle KR1.bOutBit[26,0]
        OnMouseClick: execute {  }
    Lamp1 (835,265 20x20), variable: KR1.bInBit[26,0], style: Lamp-Lamp1-Red
    RoundedRectangle (975,255 80x40), "FG1 Pos185"
        toggle KR1.bOutBit[27,2]
        OnMouseClick: execute {  }
    Lamp1 (950,265 20x20), variable: KR1.bInBit[27,2], style: Lamp-Lamp1-Red
    RoundedRectangle (1090,255 80x40), "FG1 Pos195"
        toggle KR1.bOutBit[28,4]
        OnMouseClick: execute {  }
    Lamp1 (1065,265 20x20), variable: KR1.bInBit[28,4], style: Lamp-Lamp1-Red
    RoundedRectangle (170,315 80x40), "FG1 Pos116"
        toggle KR1.bOutBit[18,5]
        OnMouseClick: execute {  }
    Lamp1 (145,325 20x20), variable: KR1.bInBit[18,5], style: Lamp-Lamp1-Red
    RoundedRectangle (55,315 80x40), "FG1 Pos106"
        toggle KR1.bOutBit[17,3]
        OnMouseClick: execute {  }
    Lamp1 (30,325 20x20), variable: KR1.bInBit[17,3], style: Lamp-Lamp1-Red
    RoundedRectangle (285,315 80x40), "FG1 Pos126"
        toggle KR1.bOutBit[19,7]
        OnMouseClick: execute {  }
    Lamp1 (260,325 20x20), variable: KR1.bInBit[19,7], style: Lamp-Lamp1-Red
    RoundedRectangle (400,315 80x40), "FG1 Pos136"
        toggle KR1.bOutBit[21,1]
        OnMouseClick: execute {  }
    Lamp1 (375,325 20x20), variable: KR1.bInBit[21,1], style: Lamp-Lamp1-Red
    RoundedRectangle (515,315 80x40), "FG1 Pos146"
        toggle KR1.bOutBit[22,3]
        OnMouseClick: execute {  }
    Lamp1 (490,325 20x20), variable: KR1.bInBit[22,3], style: Lamp-Lamp1-Red
    RoundedRectangle (745,315 80x40), "FG1 Pos166"
        toggle KR1.bOutBit[24,7]
        OnMouseClick: execute {  }
    Lamp1 (720,325 20x20), variable: KR1.bInBit[24,7], style: Lamp-Lamp1-Red
    RoundedRectangle (630,315 80x40), "FG1 Pos156"
        toggle KR1.bOutBit[23,5]
        OnMouseClick: execute {  }
    Lamp1 (605,325 20x20), variable: KR1.bInBit[23,5], style: Lamp-Lamp1-Red
    RoundedRectangle (860,315 80x40), "FG1 Pos176"
        toggle KR1.bOutBit[26,1]
        OnMouseClick: execute {  }
    Lamp1 (835,325 20x20), variable: KR1.bInBit[26,1], style: Lamp-Lamp1-Red
    RoundedRectangle (975,315 80x40), "FG1 Pos186"
        toggle KR1.bOutBit[27,3]
        OnMouseClick: execute {  }
    Lamp1 (950,325 20x20), variable: KR1.bInBit[27,3], style: Lamp-Lamp1-Red
    RoundedRectangle (1090,315 80x40), "FG1 Pos196"
        toggle KR1.bOutBit[28,5]
        OnMouseClick: execute {  }
    Lamp1 (1065,325 20x20), variable: KR1.bInBit[28,5], style: Lamp-Lamp1-Red
    RoundedRectangle (170,375 80x40), "FG1 Pos117"
        toggle KR1.bOutBit[18,6]
        OnMouseClick: execute {  }
    Lamp1 (145,385 20x20), variable: KR1.bInBit[18,6], style: Lamp-Lamp1-Red
    RoundedRectangle (55,375 80x40), "FG1 Pos107"
        toggle KR1.bOutBit[17,4]
        OnMouseClick: execute {  }
    Lamp1 (30,385 20x20), variable: KR1.bInBit[17,4], style: Lamp-Lamp1-Red
    RoundedRectangle (285,375 80x40), "FG1 Pos127"
        toggle KR1.bOutBit[20,0]
        OnMouseClick: execute {  }
    Lamp1 (260,385 20x20), variable: KR1.bInBit[20,0], style: Lamp-Lamp1-Red
    RoundedRectangle (400,375 80x40), "FG1 Pos137"
        toggle KR1.bOutBit[21,2]
        OnMouseClick: execute {  }
    Lamp1 (375,385 20x20), variable: KR1.bInBit[21,2], style: Lamp-Lamp1-Red
    RoundedRectangle (515,375 80x40), "FG1 Pos147"
        toggle KR1.bOutBit[22,4]
        OnMouseClick: execute {  }
    Lamp1 (490,385 20x20), variable: KR1.bInBit[22,4], style: Lamp-Lamp1-Red
    RoundedRectangle (745,375 80x40), "FG1 Pos167"
        toggle KR1.bOutBit[25,0]
        OnMouseClick: execute {  }
    Lamp1 (720,385 20x20), variable: KR1.bInBit[25,0], style: Lamp-Lamp1-Red
    RoundedRectangle (630,375 80x40), "FG1 Po157"
        toggle KR1.bOutBit[23,6]
        OnMouseClick: execute {  }
    Lamp1 (605,385 20x20), variable: KR1.bInBit[23,6], style: Lamp-Lamp1-Red
    RoundedRectangle (860,375 80x40), "FG1 Pos177"
        toggle KR1.bOutBit[26,2]
        OnMouseClick: execute {  }
    Lamp1 (835,385 20x20), variable: KR1.bInBit[26,2], style: Lamp-Lamp1-Red
    RoundedRectangle (975,375 80x40), "FG1 Pos187"
        toggle KR1.bOutBit[27,4]
        OnMouseClick: execute {  }
    Lamp1 (950,385 20x20), variable: KR1.bInBit[27,4], style: Lamp-Lamp1-Red
    RoundedRectangle (1090,375 80x40), "FG1 Pos197"
        toggle KR1.bOutBit[28,6]
        OnMouseClick: execute {  }
    Lamp1 (1065,385 20x20), variable: KR1.bInBit[28,6], style: Lamp-Lamp1-Red
    RoundedRectangle (170,435 80x40), "FG1 Pos118"
        toggle KR1.bOutBit[18,7]
        OnMouseClick: execute {  }
    Lamp1 (145,445 20x20), variable: KR1.bInBit[18,7], style: Lamp-Lamp1-Red
    RoundedRectangle (55,435 80x40), "FG1 Pos108"
        toggle KR1.bOutBit[17,5]
        OnMouseClick: execute {  }
    Lamp1 (30,445 20x20), variable: KR1.bInBit[17,5], style: Lamp-Lamp1-Red
    RoundedRectangle (285,435 80x40), "FG1 Pos128"
        toggle KR1.bOutBit[20,1]
        OnMouseClick: execute {  }
    Lamp1 (260,445 20x20), variable: KR1.bInBit[20,1], style: Lamp-Lamp1-Red
    RoundedRectangle (400,435 80x40), "FG1 Pos138"
        toggle KR1.bOutBit[21,3]
        OnMouseClick: execute {  }
    Lamp1 (375,445 20x20), variable: KR1.bInBit[21,3], style: Lamp-Lamp1-Red
    RoundedRectangle (515,435 80x40), "FG1 Pos148"
        toggle KR1.bOutBit[22,5]
        OnMouseClick: execute {  }
    Lamp1 (490,445 20x20), variable: KR1.bInBit[22,5], style: Lamp-Lamp1-Red
    RoundedRectangle (745,435 80x40), "FG1 Pos168"
        toggle KR1.bOutBit[25,1]
        OnMouseClick: execute {  }
    Lamp1 (720,445 20x20), variable: KR1.bInBit[25,1], style: Lamp-Lamp1-Red
    RoundedRectangle (630,435 80x40), "FG1 Pos158"
        toggle KR1.bOutBit[23,7]
        OnMouseClick: execute {  }
    Lamp1 (605,445 20x20), variable: KR1.bInBit[23,7], style: Lamp-Lamp1-Red
    RoundedRectangle (860,435 80x40), "FG1 Pos178"
        toggle KR1.bOutBit[26,3]
        OnMouseClick: execute {  }
    Lamp1 (835,445 20x20), variable: KR1.bInBit[26,3], style: Lamp-Lamp1-Red
    RoundedRectangle (975,435 80x40), "FG1 Pos188"
        toggle KR1.bOutBit[27,5]
        OnMouseClick: execute {  }
    Lamp1 (950,445 20x20), variable: KR1.bInBit[27,5], style: Lamp-Lamp1-Red
    RoundedRectangle (1090,435 80x40), "FG1 Pos198"
        toggle KR1.bOutBit[28,7]
        OnMouseClick: execute {  }
    Lamp1 (1065,445 20x20), variable: KR1.bInBit[28,7], style: Lamp-Lamp1-Red
    RoundedRectangle (55,495 80x40), "FG1 Pos109"
        toggle KR1.bOutBit[17,6]
        OnMouseClick: execute {  }
    Lamp1 (30,505 20x20), variable: KR1.bInBit[17,6], style: Lamp-Lamp1-Red
    RoundedRectangle (170,495 80x40), "FG1 Pos119"
        toggle KR1.bOutBit[19,0]
        OnMouseClick: execute {  }
    Lamp1 (145,505 20x20), variable: KR1.bInBit[19,0], style: Lamp-Lamp1-Red
    RoundedRectangle (285,495 80x40), "FG1 Pos129"
        toggle KR1.bOutBit[20,2]
        OnMouseClick: execute {  }
    Lamp1 (260,505 20x20), variable: KR1.bInBit[20,2], style: Lamp-Lamp1-Red
    RoundedRectangle (400,495 80x40), "FG1 Pos139"
        toggle KR1.bOutBit[21,4]
        OnMouseClick: execute {  }
    Lamp1 (375,505 20x20), variable: KR1.bInBit[21,4], style: Lamp-Lamp1-Red
    RoundedRectangle (515,495 80x40), "FG1 Pos149"
        toggle KR1.bOutBit[22,6]
        OnMouseClick: execute {  }
    Lamp1 (490,505 20x20), variable: KR1.bInBit[22,6], style: Lamp-Lamp1-Red
    RoundedRectangle (630,495 80x40), "FG1 Pos159"
        toggle KR1.bOutBit[24,0]
        OnMouseClick: execute {  }
    Lamp1 (605,505 20x20), variable: KR1.bInBit[24,0], style: Lamp-Lamp1-Red
    RoundedRectangle (745,495 80x40), "FG1 Pos169"
        toggle KR1.bOutBit[25,2]
        OnMouseClick: execute {  }
    Lamp1 (720,505 20x20), variable: KR1.bInBit[25,2], style: Lamp-Lamp1-Red
    RoundedRectangle (860,495 80x40), "FG1 Pos179"
        toggle KR1.bOutBit[26,4]
        OnMouseClick: execute {  }
    Lamp1 (835,505 20x20), variable: KR1.bInBit[26,4], style: Lamp-Lamp1-Red
    RoundedRectangle (975,495 80x40), "FG1 Pos189"
        toggle KR1.bOutBit[27,6]
        OnMouseClick: execute {  }
    Lamp1 (950,505 20x20), variable: KR1.bInBit[27,6], style: Lamp-Lamp1-Red
    RoundedRectangle (1090,495 80x40), "FG1 Pos199"
        toggle KR1.bOutBit[29,0]
        OnMouseClick: execute {  }
    Lamp1 (1065,505 20x20), variable: KR1.bInBit[29,0], style: Lamp-Lamp1-Red
    RoundedRectangle (55,555 80x40), "FG1 Pos110"
        toggle KR1.bOutBit[17,7]
        OnMouseClick: execute {  }
    Lamp1 (30,565 20x20), variable: KR1.bInBit[17,7], style: Lamp-Lamp1-Red
    RoundedRectangle (170,555 80x40), "FG1 Pos120"
        toggle KR1.bOutBit[19,1]
        OnMouseClick: execute {  }
    Lamp1 (145,565 20x20), variable: KR1.bInBit[19,1], style: Lamp-Lamp1-Red
    RoundedRectangle (285,555 80x40), "FG1 Pos130"
        toggle KR1.bOutBit[20,3]
        OnMouseClick: execute {  }
    Lamp1 (260,565 20x20), variable: KR1.bInBit[20,3], style: Lamp-Lamp1-Red
    RoundedRectangle (400,555 80x40), "FG1 Pos140"
        toggle KR1.bOutBit[21,5]
        OnMouseClick: execute {  }
    Lamp1 (375,565 20x20), variable: KR1.bInBit[21,5], style: Lamp-Lamp1-Red
    RoundedRectangle (515,555 80x40), "FG1 Pos150"
        toggle KR1.bOutBit[22,7]
        OnMouseClick: execute {  }
    Lamp1 (490,565 20x20), variable: KR1.bInBit[22,7], style: Lamp-Lamp1-Red
    RoundedRectangle (630,555 80x40), "FG1 Pos160"
        toggle KR1.bOutBit[24,1]
        OnMouseClick: execute {  }
    Lamp1 (605,565 20x20), variable: KR1.bInBit[24,1], style: Lamp-Lamp1-Red
    RoundedRectangle (745,555 80x40), "FG1 Pos170"
        toggle KR1.bOutBit[25,3]
        OnMouseClick: execute {  }
    Lamp1 (720,565 20x20), variable: KR1.bInBit[25,3], style: Lamp-Lamp1-Red
    RoundedRectangle (860,555 80x40), "FG1 Pos180"
        toggle KR1.bOutBit[26,5]
        OnMouseClick: execute {  }
    Lamp1 (835,565 20x20), variable: KR1.bInBit[26,5], style: Lamp-Lamp1-Red
    RoundedRectangle (975,555 80x40), "FG1 Pos190"
        toggle KR1.bOutBit[27,7]
        OnMouseClick: execute {  }
    Lamp1 (950,565 20x20), variable: KR1.bInBit[27,7], style: Lamp-Lamp1-Red
    RoundedRectangle (1090,555 80x40), "FG1 Pos200"
        toggle KR1.bOutBit[29,1]
        OnMouseClick: execute {  }
    Lamp1 (1065,565 20x20), variable: KR1.bInBit[29,1], style: Lamp-Lamp1-Red
    RoundedRectangle (55,630 80x40), "Layer pad 1"
        toggle KR1.bOutBit[29,2]
        OnMouseClick: execute {  }
    Lamp1 (30,640 20x20), variable: KR1.bInBit[29,2], style: Lamp-Lamp1-Red
    RoundedRectangle (170,630 80x40), "Layer pad 2"
        toggle KR1.bOutBit[29,3]
        OnMouseClick: execute {  }
    Lamp1 (145,640 20x20), variable: KR1.bInBit[29,3], style: Lamp-Lamp1-Red
    RoundedRectangle (285,630 80x40), "Layer pad 3"
        toggle KR1.bOutBit[29,4]
        OnMouseClick: execute {  }
    Lamp1 (260,640 20x20), variable: KR1.bInBit[29,4], style: Lamp-Lamp1-Red
    RoundedRectangle (400,630 80x40), "Layer pad 4"
        toggle KR1.bOutBit[29,5]
        OnMouseClick: execute {  }
    Lamp1 (375,640 20x20), variable: KR1.bInBit[29,5], style: Lamp-Lamp1-Red
    RoundedRectangle (515,630 80x40), "Layer pad 5"
        toggle KR1.bOutBit[29,6]
        OnMouseClick: execute {  }
    Lamp1 (490,640 20x20), variable: KR1.bInBit[29,6], style: Lamp-Lamp1-Red
    RoundedRectangle (630,630 80x40), "Layer pad 6"
        toggle KR1.bOutBit[29,7]
        OnMouseClick: execute {  }
    Lamp1 (605,640 20x20), variable: KR1.bInBit[29,7], style: Lamp-Lamp1-Red
    RoundedRectangle (745,630 80x40), "Layer pad 7"
        toggle KR1.bOutBit[30,0]
        OnMouseClick: execute {  }
    Lamp1 (720,640 20x20), variable: KR1.bInBit[30,0], style: Lamp-Lamp1-Red
    RoundedRectangle (860,630 80x40), "Layer pad 8"
        toggle KR1.bOutBit[30,1]
        OnMouseClick: execute {  }
    Lamp1 (835,640 20x20), variable: KR1.bInBit[30,1], style: Lamp-Lamp1-Red
    RoundedRectangle (975,630 80x40), "Layer pad 9"
        toggle KR1.bOutBit[30,2]
        OnMouseClick: execute {  }
    Lamp1 (950,640 20x20), variable: KR1.bInBit[30,2], style: Lamp-Lamp1-Red
    RoundedRectangle (1090,630 80x40), "Layer pad 10"
        toggle KR1.bOutBit[30,3]
        OnMouseClick: execute {  }
    Lamp1 (1065,640 20x20), variable: KR1.bInBit[30,3], style: Lamp-Lamp1-Red
END_VISUALIZATION

// ---- VISUs/PAGE_MAIN_1.TcVIS
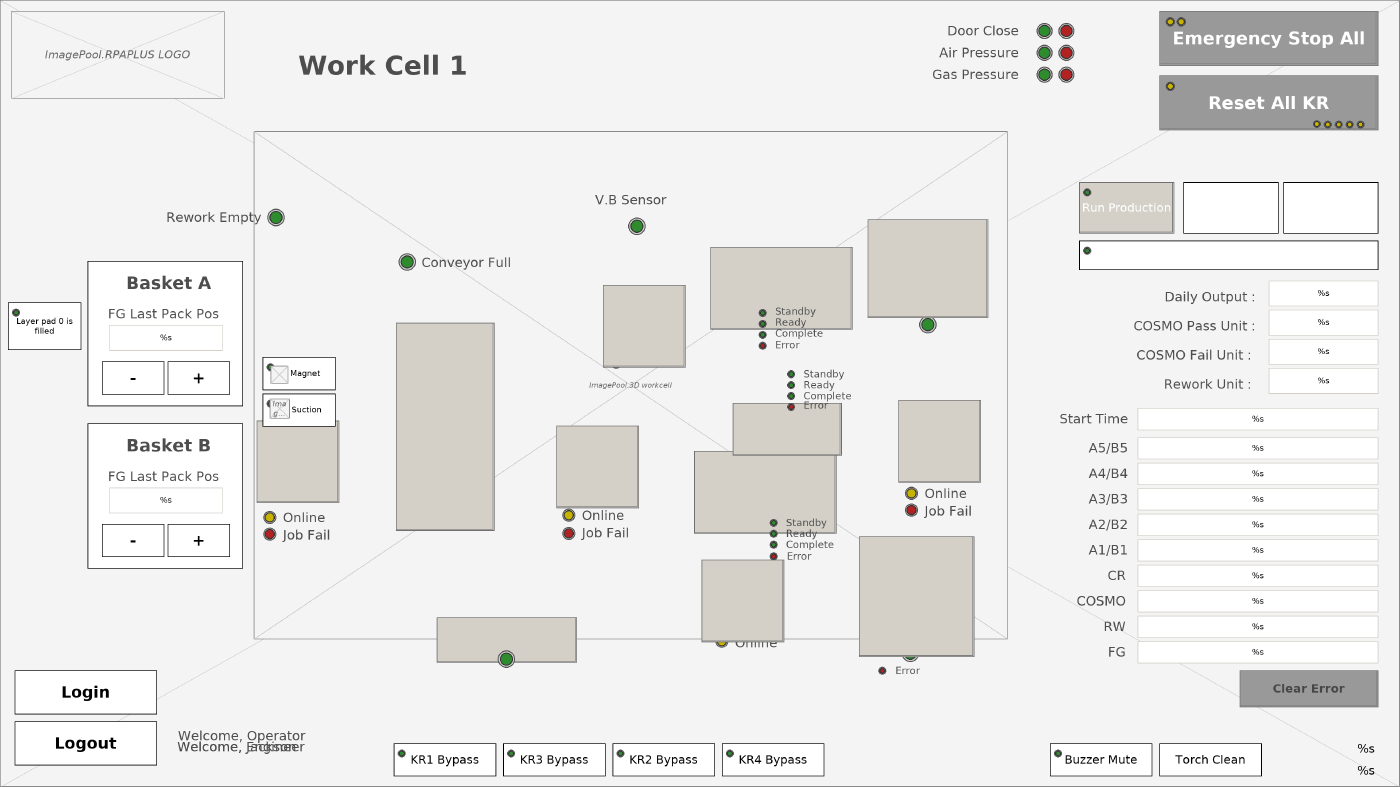
VISUALIZATION PAGE_MAIN_1  // 1920x1080
    Image (0,0 1920x1080), image: ImagePool.The-New-Silver-Backgrounds
    Frame (0,930 1920x150)
        shows Footer_Main()
        shows Footer_1()
    Frame (0,0 1920x225)
        shows Header()
    Label (300,60 450x60), "Work Cell 1"
    RoundedRectangle (1760,250 130x70), "Reset Production"
        OnMouseClick: OpenDialog Dialog=MSG_BOX_RESET, OpenModal=True, OpenCentered=True
    RoundedRectangle (20,990 195x60), "Logout"
        OnMouseClick: VisuUserMgmt Type=Logout
        OnMouseClick: execute {
            LOGFILE( sLogEvent	 := MSG.EVENT_BTN,
            		 sLogComp	 := MSG.COMP_HMI,
            		 sLogAction	 := MSG.ACTION_LOGOUT,
            	 	 logFlag	 := TRUE);
        }
    RoundedRectangle (20,920 195x60), "Login"
        tap MAIN.BTN_LOG
        OnMouseClick: VisuUserMgmt Type=Login
        OnMouseClick: execute {
            LOGFILE( sLogEvent	 := MSG.EVENT_BTN,
            		 sLogComp	 := MSG.COMP_HMI,
            		 sLogAction	 := MSG.ACTION_LOGIN,
            	 	 logFlag	 := TRUE);
        }
    Label (240,1005 200x40), "Welcome, Engineer"
    Label (240,1005 200x40), "Welcome, Jackson"
    Label (241,990 200x40), "Welcome, Operator"
    RoundedRectangle (120,358 213x199)
    Label (170,366 119x45), "Basket A"
    RoundedRectangle (140,496 85x45), "-"
        tap JIG.BasketA_Minus
        OnMouseClick: execute {
            LOGFILE( sLogEvent	 := MSG.EVENT_BTN,
            		 sLogComp	 := MSG.COMP_FG,
            		 sLogAction	 := MSG.ACTION_BSKTA_MINUS,
            	 	 logFlag	 := TRUE);
        }
    RoundedRectangle (230,496 85x45), "+"
        tap JIG.BasketA_Plus
        OnMouseClick: execute {
            LOGFILE( sLogEvent	 := MSG.EVENT_BTN,
            		 sLogComp	 := MSG.COMP_FG,
            		 sLogAction	 := MSG.ACTION_BSKTA_PLUS,
            	 	 logFlag	 := TRUE);
        }
    Textfield (150,446 155x35), "%s", text variable: GVL.Basket_A_Counter
    Label (145,416 173x30), "FG Last Pack Pos"
    RoundedRectangle (120,581 213x199)
    Label (170,589 119x45), "Basket B"
    RoundedRectangle (140,719 85x45), "-"
        tap JIG.BasketB_Minus
        OnMouseClick: execute {
            LOGFILE( sLogEvent	 := MSG.EVENT_BTN,
            		 sLogComp	 := MSG.COMP_FG,
            		 sLogAction	 := MSG.ACTION_BSKTA_MINUS,
            	 	 logFlag	 := TRUE);
        }
    RoundedRectangle (230,719 85x45), "+"
        tap JIG.BasketB_Plus
        OnMouseClick: execute {
            LOGFILE( sLogEvent	 := MSG.EVENT_BTN,
            		 sLogComp	 := MSG.COMP_FG,
            		 sLogAction	 := MSG.ACTION_BSKTB_PLUS,
            	 	 logFlag	 := TRUE);
        }
    Textfield (150,669 155x35), "%s", text variable: GVL.Basket_B_Counter
    Label (145,639 173x30), "FG Last Pack Pos"
    Image (348,180 1034x697), image: ImagePool.3D workcell
    Lamp1 (865,430 27x27), variable: KR3.bInBit[1,6], style: Lamp-Lamp1-Green
    Lamp1 (1010,815 27x27), variable: KR4.bInBit[1,6], style: Lamp-Lamp1-Green
    Lamp1 (1275,600 27x27), variable: KR5.bInBit[1,6], style: Lamp-Lamp1-Green
    Lamp1 (800,625 27x27), variable: KR2.bInBit[1,6], style: Lamp-Lamp1-Green
    Lamp1 (360,700 20x20), variable: KR1.KROnline, style: Lamp-Lamp1-Yellow
    Button (543,443 135x285)
        OnMouseClick: change screen: PAGE_CoolRack
        OnMouseClick: execute {
            LOGFILE( sLogEvent	 := MSG.EVENT_PAGE,
            		 sLogComp	 := MSG.COMP_CR,
            		 sLogAction	 := MSG.ACTION_COOLRACK,
            	 	 logFlag	 := TRUE);
        }
    Button (599,847 192x62)
        OnMouseClick: change screen: PAGE_COSMO
        OnMouseClick: execute {
            LOGFILE( sLogEvent	 := MSG.EVENT_PAGE,
            		 sLogComp	 := MSG.COMP_CM,
            		 sLogAction	 := MSG.ACTION_COSMO,
            	 	 logFlag	 := TRUE);
        }
    Lamp1 (681,891 27x27), variable: GVL.COSMO_Ready, style: Lamp-Lamp1-Green
    Lamp1 (860,297 27x27), variable: GVL.VibBowl_Ready, style: Lamp-Lamp1-Green
    Label (813,252 255x45), "V.B Sensor"
    Lamp1 (1259,432 27x27), variable: INFEED_RACK.IFRack_Ready, style: Lamp-Lamp1-Green
    Lamp1 (1235,883 27x27), variable: GVL.JIGC_Standby, style: Lamp-Lamp1-Green
    Button (1178,736 158x165)
        OnMouseClick: change screen: PAGE_TTorch
        OnMouseClick: execute {
            LOGFILE( sLogEvent	 := MSG.EVENT_PAGE,
            		 sLogComp	 := MSG.COMP_TT,
            		 sLogAction	 := MSG.ACTION_TT,
            	 	 logFlag	 := TRUE);
        }
    Button (974,339 195x113)
        OnMouseClick: change screen: PAGE_JIG_A
        OnMouseClick: execute {
            LOGFILE( sLogEvent	 := MSG.EVENT_PAGE,
            		 sLogComp	 := MSG.COMP_JIGA,
            		 sLogAction	 := MSG.ACTION_JIGA,
            	 	 logFlag	 := TRUE);
        }
    Button (952,619 195x113)
        OnMouseClick: change screen: PAGE_JIG_C
        OnMouseClick: execute {
            LOGFILE( sLogEvent	 := MSG.EVENT_PAGE,
            		 sLogComp	 := MSG.COMP_JIGC,
            		 sLogAction	 := MSG.ACTION_JIGC,
            	 	 logFlag	 := TRUE);
        }
    Button (1005,553 149x72)
        OnMouseClick: change screen: PAGE_JIG_B
        OnMouseClick: execute {
            LOGFILE( sLogEvent	 := MSG.EVENT_PAGE,
            		 sLogComp	 := MSG.COMP_JIGB,
            		 sLogAction	 := MSG.ACTION_JIGB,
            	 	 logFlag	 := TRUE);
        }
    Lamp1 (365,285 27x27), variable: GVL.Rework_Empty, style: Lamp-Lamp1-Green
    Lamp1 (545,346 27x27), variable: GVL.Conveyor_Full, style: Lamp-Lamp1-Green
    Label (225,276 146x45), "Rework Empty"
    Label (575,338 130x45), "Conveyor Full"
    Lamp1 (360,723 20x20), variable: KR1.bInBit[4,0], style: Lamp-Lamp1-Red
    Lamp1 (1240,690 20x20), variable: KR5.bInBit[4,7], style: Lamp-Lamp1-Red
    Lamp1 (770,722 20x20), variable: KR2.bInBit[3,4], style: Lamp-Lamp1-Red
    Lamp1 (395,633 27x27), variable: KR1.bInBit[1,6], style: Lamp-Lamp1-Green
    Label (385,722 80x25), "Job Fail"
    Label (385,698 80x25), "Online"
    Lamp1 (770,697 20x20), variable: KR2.KROnline, style: Lamp-Lamp1-Yellow
    Label (795,719 80x25), "Job Fail"
    Label (795,695 80x25), "Online"
    Lamp1 (1240,667 20x20), variable: KR5.KROnline, style: Lamp-Lamp1-Yellow
    Label (1265,689 80x25), "Job Fail"
    Label (1265,665 80x25), "Online"
    Lamp1 (835,487 20x20), variable: KR3.KROnline, style: Lamp-Lamp1-Yellow
    Label (860,485 80x25), "Online"
    Lamp1 (980,870 20x20), variable: KR4.KROnline, style: Lamp-Lamp1-Yellow
    Label (1005,870 80x25), "Online"
    Button (827,391 113x113)
        OnMouseClick: change screen: PAGE_KR3
        OnMouseClick: execute {
            LOGFILE( sLogEvent	 := MSG.EVENT_PAGE,
            		 sLogComp	 := MSG.COMP_KR3,
            		 sLogAction	 := MSG.ACTION_KR3,
            	 	 logFlag	 := TRUE);
        }
    Button (763,584 113x113)
        OnMouseClick: change screen: PAGE_KR2
        OnMouseClick: execute {
            LOGFILE( sLogEvent	 := MSG.EVENT_PAGE,
            		 sLogComp	 := MSG.COMP_KR2,
            		 sLogAction	 := MSG.ACTION_KR2,
            	 	 logFlag	 := TRUE);
        }
    Button (962,768 113x113)
        OnMouseClick: change screen: PAGE_KR4
        OnMouseClick: execute {
            LOGFILE( sLogEvent	 := MSG.EVENT_PAGE,
            		 sLogComp	 := MSG.COMP_KR4,
            		 sLogAction	 := MSG.ACTION_KR4,
            	 	 logFlag	 := TRUE);
        }
    Button (1232,549 113x113)
        OnMouseClick: change screen: PAGE_KR5
        OnMouseClick: execute {
            LOGFILE( sLogEvent	 := MSG.EVENT_PAGE,
            		 sLogComp	 := MSG.COMP_KR5,
            		 sLogAction	 := MSG.ACTION_KR5,
            	 	 logFlag	 := TRUE);
        }
    Button (352,577 113x113)
        OnMouseClick: change screen: PAGE_KR1_Tab
        OnMouseClick: execute {
            LOGFILE( sLogEvent	 := MSG.EVENT_PAGE,
            		 sLogComp	 := MSG.COMP_KR1,
            		 sLogAction	 := MSG.ACTION_KR1,
            	 	 logFlag	 := TRUE);
        }
    Label (1500,425 225x45), "COSMO Pass Unit :"
    Textfield (1740,425 150x35), "%s", text variable: GVL.Pass_Counter
    Textfield (1740,465 150x35), "%s", text variable: GVL.Fail_Counter
    Label (1500,465 225x45), "COSMO Fail Unit :"
    Textfield (1560,880 330x30), "%s", text variable: AUTO_MODE.processnameFG
    Group (1430,705 460x30)
        Textfield (130,0 330x30), "%s", text variable: AUTO_MODE.processnameA2
        Label (0,0 120x30), "A2/B2"
    Group (1430,740 460x30)
        Textfield (130,0 330x30), "%s", text variable: AUTO_MODE.processnameA1
        Label (0,0 120x30), "A1/B1"
    Textfield (1560,600 330x30), "%s", text variable: AUTO_MODE.processnameA5
    Label (1430,600 120x30), "A5/B5"
    Group (1430,635 460x30)
        Textfield (130,0 330x30), "%s", text variable: AUTO_MODE.processnameA4
        Label (0,0 120x30), "A4/B4"
    Group (1430,670 460x30)
        Textfield (130,0 330x30), "%s", text variable: AUTO_MODE.processnameA3
        Label (0,0 120x30), "A3/B3"
    Label (1472,880 75x30), "FG"
    Group (1472,845 418x30)
        Textfield (88,0 330x30), "%s", text variable: AUTO_MODE.processnameRW
        Label (0,0 75x30), "RW"
    Group (1472,775 418x30)
        Textfield (88,0 330x30), "%s", text variable: AUTO_MODE.processnameCR
        Label (0,0 75x30), "CR"
    Group (1455,810 435x30)
        Textfield (105,0 330x30), "%s", text variable: AUTO_MODE.processnameCOSMO
        Label (0,0 92x30), "COSMO"
    Lamp1 (1260,358 20x20), variable: INFEED_RACK.IFRack_Ready, style: Lamp-Lamp1-Yellow
    Button (1190,301 165x135)
        OnMouseClick: change screen: PAGE_InfeedRack
        OnMouseClick: execute {
            LOGFILE( sLogEvent	 := MSG.EVENT_PAGE,
            		 sLogComp	 := MSG.COMP_IR,
            		 sLogAction	 := MSG.ACTION_INFEEDRACK,
            	 	 logFlag	 := TRUE);
        }
    Label (1500,385 225x45), "Daily Output :"
    Textfield (1740,385 150x35), "%s", text variable: GVL.daily_output
    Label (1500,505 225x45), "Rework Unit :"
    Textfield (1740,505 150x35), "%s", text variable: GVL.Rework_Counter
    RoundedRectangle (1480,330 410x40), "Welding Mode"
        toggle SAFETY_SENSOR.WELDING_MODE
        OnMouseClick: execute {  }
    RoundedRectangle (1623,250 130x70), "Halt Production", input disabled if: MAIN.btnTorchClean
        OnMouseClick: execute {
            KR1.bOutBit[1,0]:= FALSE;
            KR2.bOutBit[1,0]:= FALSE;
            KR3.bOutBit[1,0]:= FALSE;
            KR4.bOutBit[1,0]:= FALSE;
            KR5.bOutBit[1,0]:= FALSE;
            LOGFILE( sLogEvent	 := MSG.EVENT_BTN,
            		 sLogComp	 := MSG.COMP_HMI,
            		 sLogAction	 := MSG.ACTION_STOP,
            	 	 logFlag	 := TRUE);
            AUTO_MODE.Halt_Production := TRUE;
            AUTO_MODE.AutoMode := False;
        }
    Button (1480,250 130x70), "Run Production", pressed state: AUTO_MODE.AutoMode, input disabled if: MAIN.btnTorchClean
        toggle AUTO_MODE.AutoMode
        OnMouseClick: execute {
            LOGFILE( sLogEvent	 := MSG.EVENT_BTN,
            		 sLogComp	 := MSG.COMP_HMI,
            		 sLogAction	 := MSG.ACTION_START,
            	 	 logFlag	 := TRUE);
            IF AUTO_MODE.AutoMode THEN
            	AUTO_MODE.Start_time := MAIN.fb_TimeStamp.SystemTime;
            END_IF
        }
    Lamp1 (1485,255 12x18), variable: AUTO_MODE.AutoMode, style: Lamp-Lamp1-Green
    Textfield (1560,560 330x30), "%s", text variable: AUTO_MODE.Start_time
    Label (1430,560 120x30), "Start Time"
    Lamp1 (1485,335 12x18), variable: SAFETY_SENSOR.WELDING_MODE, style: Lamp-Lamp1-Green
    Group (1250,20 225x105)
        Group (0,0 225x45)
            Label (0,0 150x45), "Door Close"
            Lamp1 (170,10 25x25), variable: SAFETY_SENSOR.SENSOR_SAFETY_DOOR_CLOSE, style: Lamp-Lamp1-Green
            Lamp1 (200,10 25x25), variable: not SAFETY_SENSOR.SENSOR_SAFETY_DOOR_CLOSE, style: Lamp-Lamp1-Red
        Label (0,30 150x45), "Air Pressure"
        Lamp1 (170,40 25x25), variable: SAFETY_SENSOR.SENSOR_AIR_PRESSURE_OK, style: Lamp-Lamp1-Green
        Lamp1 (200,40 25x25), variable: not SAFETY_SENSOR.SENSOR_AIR_PRESSURE_OK or SAFETY_SENSOR.SENSOR_AIR_PRESSURE_HIGH, style: Lamp-Lamp1-Red
        Label (0,60 150x45), "Gas Pressure"
        Lamp1 (170,70 25x25), variable: SAFETY_SENSOR.SENSOR_GAS_PRESSURE_OK, style: Lamp-Lamp1-Green
        Lamp1 (200,70 25x25), variable: not SAFETY_SENSOR.SENSOR_GAS_PRESSURE_OK or SAFETY_SENSOR.SENSOR_GAS_PRESSURE_HIGH, style: Lamp-Lamp1-Red
    Group (1079,506 100x45)
        Lamp1 (0,0 12x15), variable: GVL.JIGB_Standby, style: Lamp-Lamp1-Green
        Lamp1 (0,15 12x15), variable: GVL.JIGB_Ready, style: Lamp-Lamp1-Green
        Label (20,0 80x15), "Standby"
        Label (20,15 80x15), "Ready"
        Label (20,30 80x15), "Complete"
        Lamp1 (0,30 12x15), variable: GVL.JIGB_Complete, style: Lamp-Lamp1-Green
    Lamp1 (1040,422 12x15), variable: GVL.JIGA_Standby, style: Lamp-Lamp1-Green
    Lamp1 (1040,437 12x15), variable: GVL.JIGA_Ready, style: Lamp-Lamp1-Green
    Label (1060,420 80x15), "Standby"
    Label (1060,435 80x15), "Ready"
    Label (1060,450 80x15), "Complete"
    Lamp1 (1040,452 12x15), variable: GVL.JIGA_Complete, style: Lamp-Lamp1-Green
    Lamp1 (1055,710 12x15), variable: GVL.JIGC_Standby, style: Lamp-Lamp1-Green
    Lamp1 (1055,725 12x15), variable: GVL.JIGC_Ready, style: Lamp-Lamp1-Green
    Label (1075,710 80x15), "Standby"
    Label (1075,725 80x15), "Ready"
    Label (1075,740 80x15), "Complete"
    Lamp1 (1055,740 12x15), variable: GVL.JIGC_Complete, style: Lamp-Lamp1-Green
    Button (1700,920 190x50), "Clear Error", pressed state: MAIN.btn_Reset or MAIN.Reset_State
        toggle GVL.ClearError
        OnMouseClick: execute {
            LOGFILE( sLogEvent	 := MSG.EVENT_BTN,
            		 sLogComp	 := MSG.COMP_HMI,
            		 sLogAction	 := MSG.ACTION_CLEAR_ERROR,
            	 	 logFlag	 := TRUE);
        }
    Label (1060,466 80x15), "Error"
    Lamp1 (1040,467 12x15), variable: AUTO_MODE.JIGA_ErrorState, style: Lamp-Lamp1-Red
    Lamp1 (1079,551 12x15), variable: AUTO_MODE.JIGB_ErrorState, style: Lamp-Lamp1-Red
    Label (1099,549 80x15), "Error"
    Lamp1 (1055,756 12x15), variable: AUTO_MODE.JIGC_ErrorState, style: Lamp-Lamp1-Red
    Label (1076,756 80x15), "Error"
    Lamp1 (1204,913 12x15), variable: AUTO_MODE.TT_ErrorState, style: Lamp-Lamp1-Red
    Label (1225,913 80x15), "Error"
    RoundedRectangle (1590,1020 140x45), "Torch Clean"
        toggle MAIN.btnTorchClean
        OnMouseClick: execute {  }
    Group (1440,1020 140x45)
        RoundedRectangle (0,0 140x45), "Buzzer Mute"
            toggle TL.Buzzer_mute
            OnMouseClick: execute {  }
        Lamp1 (5,5 12x18), variable: TL.Buzzer_mute, style: Lamp-Lamp1-Green
    Group (840,1020 290x45)
        Group (150,0 140x45)
            RoundedRectangle (0,0 140x45), "KR4 Bypass"
                OnMouseClick: OpenDialog Dialog=MSG_KR4_BP, OpenModal=True, OpenCentered=True
            Lamp1 (5,5 12x18), variable: GVL.KR4_bypass, style: Lamp-Lamp1-Green
        RoundedRectangle (0,0 140x45), "KR2 Bypass"
            OnMouseClick: OpenDialog Dialog=MSG_KR2_BP, OpenModal=True, OpenCentered=True
        Lamp1 (5,5 12x18), variable: GVL.KR2_bypass, style: Lamp-Lamp1-Green
    RoundedRectangle (690,1020 140x45), "KR3 Bypass"
        OnMouseClick: OpenDialog Dialog=MSG_KR3_BP, OpenModal=True, OpenCentered=True
    Lamp1 (695,1025 12x18), variable: GVL.KR3_bypass, style: Lamp-Lamp1-Green
    RoundedRectangle (540,1020 140x45), "KR1 Bypass"
        OnMouseClick: OpenDialog Dialog=MSG_KR1_BP, OpenModal=True, OpenCentered=True
    Lamp1 (545,1025 12x18), variable: GVL.KR1_bypass, style: Lamp-Lamp1-Green
    Group (360,490 100x45)
        RoundedRectangle (0,0 100x45), "Magnet"
            OnMouseClick: OpenDialog Dialog=MSG_EOAT, OpenModal=True, OpenCentered=True
        Lamp1 (5,5 12x18), variable: GVL.KR1_EOAT_FILL, style: Lamp-Lamp1-Green
        Image (11,12 24x24), image: ImagePool.001-resources
    Group (360,540 100x45)
        RoundedRectangle (0,0 100x45), "Suction"
            OnMouseClick: OpenDialog Dialog=MSG_EOAT_SUCTION, OpenModal=True, OpenCentered=True
        Lamp1 (5,5 12x18), variable: GVL.KR1_EOAT_SUCTION, style: Lamp-Lamp1-Green
        Image (10,7 27x27), angle 180, image: ImagePool.002-plunger
    RoundedRectangle (11,415 100x65), "Layer pad 0 is filled"
        toggle GVL.LAYERPAD0
    Lamp1 (16,420 12x18), variable: GVL.LAYERPAD0, style: Lamp-Lamp1-Green
END_VISUALIZATION

// ---- VISUs/PAGE_TTorch.TcVIS
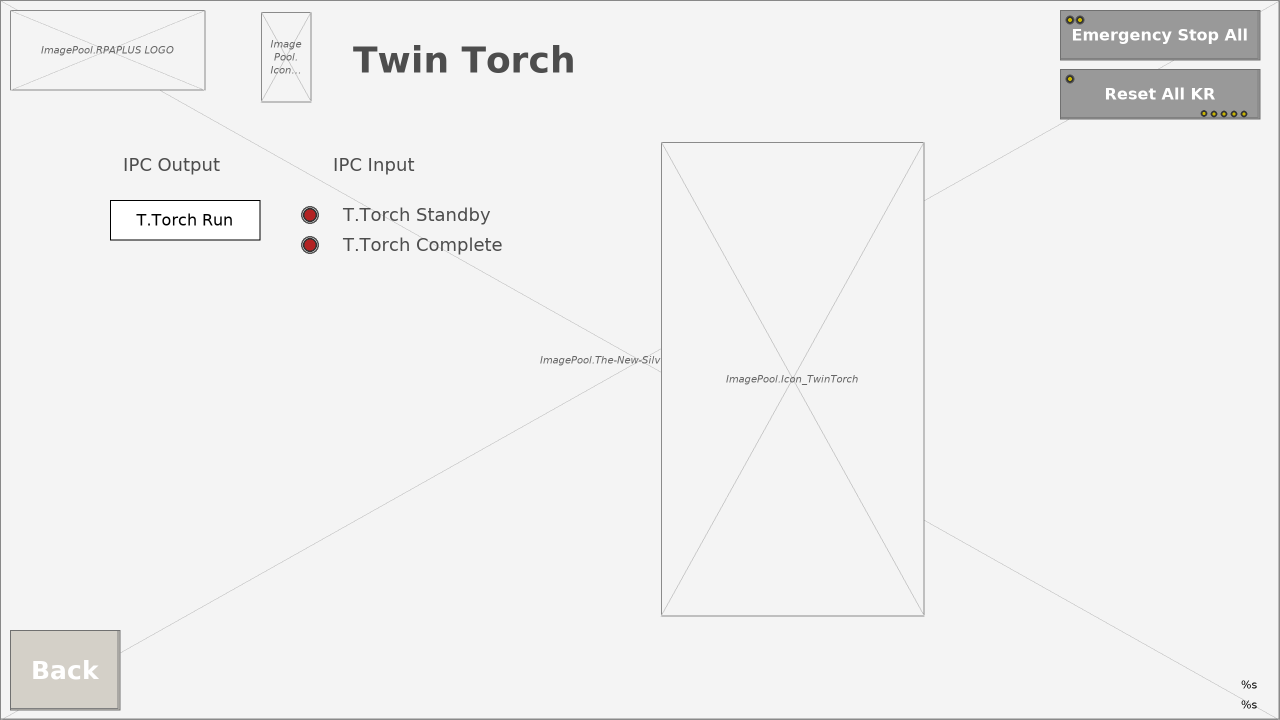
VISUALIZATION PAGE_TTorch  // 1280x720
    Image (0,0 1280x720), image: ImagePool.The-New-Silver-Backgrounds
    Frame (0,620 1280x100)
        shows Footer_Back()
    Frame (0,0 1280x150)
        shows Header()
    Label (350,40 300x40), "Twin Torch"
    Label (120,150 150x30), "IPC Output"
    RoundedRectangle (110,200 150x40), "T.Torch Run"
        toggle GVL.TTorch_Run
    Label (330,150 150x30), "IPC Input"
    Label (340,200 170x30), "T.Torch Standby"
    Lamp1 (300,205 20x20), variable: GVL.TTorch_Standy, style: Lamp-Lamp1-Red
    Label (340,230 170x30), "T.Torch Complete"
    Lamp1 (300,235 20x20), variable: GVL.TTorch_Complete, style: Lamp-Lamp1-Red
    Image (261,12 50x90), image: ImagePool.Icon_TwinTorch
    Image (661,142 263x474), image: ImagePool.Icon_TwinTorch
END_VISUALIZATION

